C05459=1044.843,173.634,405.033,170.769,37.953,157.158
C05460=1044.836,173.349,405.060,170.766,37.951,157.157
C05461=1044.829,173.064,405.087,170.763,37.949,157.157
C05462=1044.823,172.815,405.109,170.761,37.947,157.156
C05463=1044.817,172.567,405.132,170.759,37.946,157.156
C05464=1044.810,172.318,405.156,170.756,37.945,157.156
C05465=1044.804,172.069,405.179,170.754,37.943,157.155
C05466=1044.799,171.820,405.202,170.752,37.942,157.155
C05467=1044.793,171.572,405.226,170.749,37.940,157.155
C05468=1044.787,171.323,405.249,170.747,37.938,157.154
C05469=1044.780,171.073,405.272,170.744,37.937,157.154
C05470=1044.774,170.824,405.295,170.742,37.935,157.154
C05471=1044.768,170.576,405.318,170.739,37.933,157.153
C05472=1044.762,170.327,405.341,170.737,37.932,157.153
C05473=1044.757,170.078,405.364,170.735,37.930,157.153
C05474=1044.750,169.829,405.387,170.733,37.929,157.152
C05475=1044.744,169.580,405.410,170.730,37.927,157.152
C05476=1044.738,169.331,405.433,170.728,37.926,157.151
C05477=1044.732,169.083,405.456,170.726,37.925,157.151
C05478=1044.726,168.834,405.479,170.723,37.923,157.151
C05479=1044.720,168.585,405.503,170.721,37.921,157.150
C05480=1044.714,168.336,405.526,170.719,37.920,157.150
C05481=1044.708,168.087,405.548,170.717,37.918,157.150
C05482=1044.702,167.838,405.571,170.714,37.916,157.149
C05483=1044.696,167.589,405.594,170.712,37.915,157.149
C05484=1044.690,167.341,405.617,170.709,37.913,157.149
C05485=1044.685,167.092,405.640,170.707,37.912,157.148
C05486=1044.679,166.843,405.663,170.704,37.910,157.148
C05487=1044.672,166.594,405.686,170.702,37.909,157.148
C05488=1044.666,166.345,405.709,170.700,37.907,157.147
C05489=1044.660,166.096,405.732,170.697,37.906,157.147
C05490=1044.655,165.847,405.755,170.695,37.904,157.147
C05491=1044.649,165.598,405.778,170.693,37.903,157.146
C05492=1044.642,165.350,405.800,170.691,37.901,157.146
C05493=1044.637,165.101,405.823,170.688,37.900,157.146
C05494=1044.631,164.852,405.846,170.686,37.898,157.145
C05495=1044.625,164.603,405.869,170.684,37.896,157.145
C05496=1044.619,164.354,405.892,170.682,37.895,157.145
C05497=1044.613,164.106,405.914,170.679,37.893,157.144
C05498=1044.607,163.857,405.937,170.677,37.891,157.144
C05499=1044.601,163.607,405.961,170.675,37.890,157.144
C05500=1044.595,163.358,405.984,170.672,37.889,157.143
C05501=1044.589,163.109,406.007,170.670,37.887,157.143
C05502=1044.583,162.861,406.029,170.668,37.886,157.143
C05503=1044.577,162.612,406.052,170.666,37.884,157.142
C05504=1044.572,162.363,406.075,170.663,37.883,157.142
C05505=1044.566,162.114,406.098,170.661,37.881,157.142
C05506=1044.560,161.865,406.119,170.659,37.879,157.141
C05507=1044.554,161.616,406.142,170.657,37.878,157.141
C05508=1044.548,161.367,406.165,170.654,37.876,157.140
C05509=1044.542,161.118,406.188,170.652,37.875,157.140
C05510=1044.537,160.869,406.211,170.650,37.873,157.140
C05511=1044.530,160.621,406.233,170.647,37.871,157.139
C05512=1044.525,160.372,406.256,170.645,37.870,157.139
C05513=1044.519,160.122,406.279,170.643,37.868,157.139
C05514=1044.513,159.874,406.301,170.641,37.867,157.138
C05515=1044.506,159.625,406.323,170.638,37.865,157.138
C05516=1044.501,159.376,406.346,170.636,37.864,157.138
C05517=1044.494,159.127,406.368,170.634,37.863,157.138
C05518=1044.489,158.878,406.391,170.632,37.861,157.137
C05519=1044.482,158.629,406.413,170.629,37.860,157.137
C05520=1044.476,158.380,406.435,170.627,37.858,157.137
C05521=1044.470,158.131,406.458,170.625,37.857,157.136
C05522=1044.463,157.846,406.483,170.623,37.855,157.136
C05523=1044.456,157.561,406.509,170.620,37.854,157.136
C05524=1044.449,157.275,406.534,170.617,37.852,157.135
C05525=1044.441,156.990,406.560,170.615,37.851,157.135
C05526=1044.436,156.741,406.582,170.613,37.850,157.135
C05527=1044.430,156.492,406.605,170.610,37.848,157.134
C05528=1044.423,156.243,406.626,170.608,37.847,157.134
C05529=1044.418,155.994,406.649,170.606,37.845,157.134
C05530=1044.411,155.745,406.672,170.604,37.844,157.133
C05531=1044.405,155.496,406.693,170.601,37.842,157.133
C05532=1044.400,155.248,406.716,170.599,37.841,157.133
C05533=1044.394,154.999,406.738,170.597,37.839,157.132
C05534=1044.388,154.750,406.761,170.595,37.838,157.132
C05535=1044.382,154.501,406.782,170.592,37.837,157.132
C05536=1044.375,154.252,406.804,170.590,37.835,157.131
C05537=1044.369,154.003,406.826,170.588,37.834,157.131
C05538=1044.363,153.754,406.849,170.586,37.832,157.131
C05539=1044.357,153.505,406.871,170.583,37.831,157.131
C05540=1044.351,153.256,406.893,170.581,37.829,157.130
C05541=1044.345,153.007,406.915,170.579,37.828,157.130
C05542=1044.338,152.758,406.937,170.577,37.827,157.130
C05543=1044.333,152.509,406.959,170.574,37.825,157.129
C05544=1044.326,152.260,406.982,170.572,37.824,157.129
C05545=1044.320,152.011,407.003,170.570,37.823,157.129
C05546=1044.314,151.762,407.026,170.569,37.821,157.128
C05547=1044.308,151.513,407.048,170.567,37.820,157.128
C05548=1044.302,151.264,407.069,170.564,37.819,157.128
C05549=1044.296,151.016,407.091,170.562,37.817,157.127
C05550=1044.290,150.767,407.113,170.560,37.816,157.127
C05551=1044.284,150.518,407.135,170.558,37.815,157.127
C05552=1044.278,150.269,407.158,170.555,37.813,157.126
C05553=1044.272,150.019,407.179,170.553,37.812,157.126
C05554=1044.266,149.771,407.202,170.551,37.810,157.126
C05555=1044.259,149.522,407.223,170.549,37.809,157.126
C05556=1044.253,149.272,407.245,170.546,37.808,157.125
C05557=1044.247,149.024,407.267,170.544,37.806,157.125
C05558=1044.242,148.775,407.289,170.542,37.805,157.125
C05559=1044.236,148.526,407.311,170.540,37.803,157.124
C05560=1044.230,148.277,407.332,170.538,37.802,157.124
C05561=1044.223,148.028,407.355,170.535,37.801,157.124
C05562=1044.217,147.779,407.376,170.533,37.799,157.123
C05563=1044.211,147.530,407.398,170.532,37.798,157.123
C05564=1044.205,147.280,407.420,170.530,37.797,157.123
C05565=1044.199,147.032,407.442,170.527,37.796,157.123
C05566=1044.193,146.783,407.463,170.525,37.794,157.122
C05567=1044.186,146.534,407.485,170.523,37.793,157.122
C05568=1044.180,146.285,407.507,170.521,37.792,157.122
C05569=1044.174,146.036,407.528,170.518,37.790,157.122
C05570=1044.168,145.787,407.551,170.516,37.789,157.121
C05571=1044.161,145.538,407.572,170.514,37.787,157.121
C05572=1044.156,145.289,407.593,170.512,37.786,157.121
C05573=1044.150,145.040,407.615,170.510,37.785,157.120
C05574=1044.144,144.791,407.637,170.507,37.784,157.120
C05575=1044.137,144.542,407.658,170.505,37.783,157.120
C05576=1044.131,144.293,407.680,170.503,37.781,157.119
C05577=1044.125,144.045,407.702,170.502,37.780,157.119
C05578=1044.119,143.795,407.724,170.499,37.778,157.119
C05579=1044.113,143.546,407.745,170.497,37.777,157.119
C05580=1044.107,143.297,407.767,170.495,37.775,157.118
C05581=1044.101,143.048,407.789,170.493,37.774,157.118
C05582=1044.095,142.799,407.810,170.491,37.773,157.118
C05583=1044.089,142.550,407.831,170.488,37.772,157.117
C05584=1044.082,142.301,407.852,170.486,37.771,157.117
C05585=1044.076,142.052,407.874,170.484,37.769,157.117
C05586=1044.069,141.767,407.899,170.482,37.768,157.117
C05587=1044.063,141.481,407.924,170.479,37.766,157.116
C05588=1044.056,141.195,407.949,170.477,37.765,157.116
C05589=1044.048,140.909,407.973,170.475,37.763,157.116
C05590=1044.043,140.661,407.994,170.473,37.762,157.115
C05591=1044.037,140.412,408.016,170.470,37.761,157.115
C05592=1044.030,140.162,408.037,170.468,37.759,157.115
C05593=1044.024,139.913,408.059,170.466,37.758,157.114
C05594=1044.019,139.665,408.080,170.464,37.757,157.114
C05595=1044.013,139.416,408.102,170.462,37.755,157.114
C05596=1044.006,139.166,408.123,170.459,37.754,157.114
C05597=1043.999,138.917,408.144,170.458,37.753,157.113
C05598=1043.994,138.669,408.166,170.456,37.751,157.113
C05599=1043.988,138.420,408.187,170.454,37.750,157.113
C05600=1043.982,138.170,408.209,170.451,37.749,157.112
C05601=1043.975,137.922,408.230,170.449,37.748,157.112
C05602=1043.969,137.672,408.251,170.447,37.746,157.112
C05603=1043.963,137.423,408.272,170.445,37.745,157.112
C05604=1043.957,137.174,408.294,170.443,37.744,157.111
C05605=1043.951,136.926,408.315,170.441,37.742,157.111
C05606=1043.945,136.677,408.336,170.439,37.741,157.111
C05607=1043.939,136.427,408.357,170.437,37.740,157.110
C05608=1043.933,136.179,408.378,170.435,37.739,157.110
C05609=1043.926,135.929,408.399,170.433,37.737,157.110
C05610=1043.920,135.680,408.421,170.430,37.736,157.110
C05611=1043.914,135.431,408.443,170.428,37.735,157.109
C05612=1043.908,135.182,408.463,170.426,37.734,157.109
C05613=1043.902,134.933,408.484,170.425,37.733,157.109
C05614=1043.896,134.684,408.506,170.422,37.731,157.109
C05615=1043.889,134.436,408.527,170.420,37.730,157.108
C05616=1043.884,134.186,408.547,170.418,37.729,157.108
C05617=1043.878,133.937,408.569,170.416,37.727,157.108
C05618=1043.871,133.688,408.590,170.414,37.726,157.107
C05619=1043.865,133.439,408.611,170.411,37.725,157.107
C05620=1043.860,133.190,408.632,170.410,37.724,157.107
C05621=1043.853,132.941,408.653,170.408,37.723,157.107
C05622=1043.847,132.692,408.675,170.406,37.721,157.106
C05623=1043.841,132.443,408.695,170.404,37.720,157.106
C05624=1043.834,132.194,408.716,170.401,37.718,157.106
C05625=1043.828,131.945,408.738,170.399,37.717,157.106
C05626=1043.823,131.696,408.758,170.397,37.716,157.105
C05627=1043.816,131.447,408.779,170.396,37.715,157.105
C05628=1043.811,131.198,408.800,170.394,37.714,157.105
C05629=1043.804,130.949,408.821,170.391,37.712,157.104
C05630=1043.798,130.699,408.843,170.389,37.711,157.104
C05631=1043.792,130.451,408.863,170.387,37.710,157.104
C05632=1043.785,130.202,408.884,170.385,37.709,157.104
C05633=1043.779,129.952,408.905,170.383,37.708,157.103
C05634=1043.773,129.704,408.925,170.381,37.707,157.103
C05635=1043.767,129.454,408.946,170.379,37.705,157.103
C05636=1043.760,129.205,408.967,170.377,37.704,157.103
C05637=1043.754,128.956,408.987,170.375,37.703,157.102
C05638=1043.748,128.707,409.009,170.373,37.702,157.102
C05639=1043.742,128.458,409.029,170.370,37.701,157.102
C05640=1043.735,128.209,409.050,170.368,37.699,157.102
C05641=1043.729,127.959,409.071,170.367,37.698,157.101
C05642=1043.723,127.711,409.091,170.365,37.697,157.101
C05643=1043.716,127.462,409.112,170.363,37.696,157.101
C05644=1043.711,127.213,409.132,170.360,37.695,157.101
C05645=1043.704,126.964,409.153,170.358,37.693,157.100
C05646=1043.698,126.714,409.174,170.356,37.692,157.100
C05647=1043.692,126.466,409.195,170.354,37.691,157.100
C05648=1043.685,126.216,409.215,170.353,37.690,157.100
C05649=1043.680,125.967,409.236,170.350,37.689,157.099
C05650=1043.672,125.681,409.260,170.348,37.687,157.099
C05651=1043.665,125.396,409.284,170.346,37.686,157.099
C05652=1043.658,125.110,409.308,170.343,37.685,157.098
C05653=1043.651,124.824,409.331,170.341,37.683,157.098
C05654=1043.645,124.575,409.351,170.339,37.682,157.098
C05655=1043.639,124.325,409.372,170.337,37.681,157.098
C05656=1043.633,124.077,409.393,170.335,37.680,157.097
C05657=1043.626,123.828,409.413,170.333,37.679,157.097
C05658=1043.620,123.578,409.434,170.331,37.677,157.097
C05659=1043.614,123.330,409.455,170.328,37.676,157.097
C05660=1043.607,123.080,409.475,170.327,37.675,157.096
C05661=1043.602,122.831,409.496,170.325,37.674,157.096
C05662=1043.595,122.582,409.516,170.323,37.673,157.096
C05663=1043.589,122.333,409.537,170.321,37.671,157.096
C05664=1043.583,122.085,409.557,170.318,37.670,157.095
C05665=1043.577,121.835,409.577,170.317,37.669,157.095
C05666=1043.571,121.587,409.598,170.315,37.668,157.095
C05667=1043.564,121.337,409.618,170.313,37.667,157.095
C05668=1043.559,121.088,409.639,170.311,37.665,157.094
C05669=1043.553,120.838,409.659,170.308,37.664,157.094
C05670=1043.547,120.590,409.679,170.307,37.663,157.094
C05671=1043.540,120.340,409.701,170.305,37.662,157.093
C05672=1043.534,120.092,409.721,170.303,37.661,157.093
C05673=1043.528,119.842,409.741,170.301,37.659,157.093
C05674=1043.523,119.593,409.762,170.298,37.658,157.093
C05675=1043.516,119.345,409.782,170.297,37.657,157.092
C05676=1043.510,119.095,409.803,170.295,37.656,157.092
C05677=1043.504,118.846,409.823,170.293,37.655,157.092
C05678=1043.498,118.597,409.844,170.291,37.653,157.092
C05679=1043.492,118.348,409.864,170.288,37.652,157.091
C05680=1043.485,118.098,409.884,170.287,37.651,157.091
C05681=1043.480,117.849,409.904,170.285,37.650,157.091
C05682=1043.474,117.601,409.925,170.283,37.649,157.091
C05683=1043.467,117.351,409.945,170.281,37.647,157.090
C05684=1043.461,117.103,409.965,170.280,37.646,157.090
C05685=1043.456,116.854,409.986,170.277,37.645,157.090
C05686=1043.449,116.604,410.006,170.275,37.644,157.090
C05687=1043.443,116.355,410.026,170.273,37.643,157.089
C05688=1043.437,116.105,410.047,170.271,37.641,157.089
C05689=1043.431,115.857,410.067,170.269,37.640,157.089
C05690=1043.425,115.608,410.087,170.267,37.638,157.088
C05691=1043.419,115.358,410.107,170.265,37.637,157.088
C05692=1043.413,115.110,410.129,170.263,37.636,157.088
C05693=1043.407,114.861,410.149,170.262,37.635,157.088
C05694=1043.401,114.611,410.169,170.259,37.634,157.087
C05695=1043.395,114.363,410.189,170.257,37.632,157.087
C05696=1043.389,114.113,410.209,170.255,37.631,157.087
C05697=1043.383,113.864,410.230,170.254,37.630,157.087
C05698=1043.377,113.615,410.250,170.252,37.629,157.086
C05699=1043.371,113.366,410.270,170.250,37.628,157.086
C05700=1043.364,113.117,410.290,170.247,37.626,157.086
C05701=1043.358,112.868,410.310,170.246,37.625,157.086
C05702=1043.353,112.619,410.329,170.244,37.624,157.085
C05703=1043.346,112.369,410.350,170.242,37.623,157.085
C05704=1043.340,112.120,410.370,170.240,37.622,157.085
C05705=1043.333,111.871,410.390,170.237,37.621,157.085
C05706=1043.327,111.622,410.410,170.236,37.620,157.085
C05707=1043.321,111.373,410.430,170.234,37.619,157.084
C05708=1043.315,111.124,410.450,170.232,37.617,157.084
C05709=1043.309,110.875,410.470,170.230,37.616,157.084
C05710=1043.303,110.626,410.490,170.228,37.615,157.083
C05711=1043.296,110.376,410.510,170.226,37.614,157.083
C05712=1043.290,110.127,410.530,170.224,37.613,157.083
C05713=1043.284,109.878,410.550,170.222,37.611,157.083
C05714=1043.278,109.592,410.572,170.220,37.610,157.082
C05715=1043.270,109.306,410.595,170.218,37.609,157.082
C05716=1043.263,109.020,410.618,170.215,37.608,157.082
C05717=1043.256,108.734,410.640,170.213,37.607,157.082
C05718=1043.250,108.485,410.660,170.211,37.605,157.081
C05719=1043.243,108.236,410.681,170.209,37.604,157.081
C05720=1043.237,107.986,410.700,170.208,37.603,157.081
C05721=1043.231,107.737,410.720,170.205,37.602,157.081
C05722=1043.224,107.488,410.740,170.203,37.601,157.081
C05723=1043.218,107.239,410.760,170.201,37.600,157.080
C05724=1043.212,106.990,410.779,170.200,37.599,157.080
C05725=1043.206,106.741,410.799,170.198,37.598,157.080
C05726=1043.200,106.492,410.819,170.195,37.596,157.079
C05727=1043.194,106.243,410.839,170.193,37.595,157.079
C05728=1043.188,105.993,410.858,170.192,37.594,157.079
C05729=1043.181,105.745,410.878,170.190,37.593,157.079
C05730=1043.175,105.495,410.898,170.188,37.592,157.079
C05731=1043.169,105.246,410.917,170.186,37.591,157.078
C05732=1043.163,104.997,410.937,170.183,37.590,157.078
C05733=1043.157,104.748,410.957,170.182,37.589,157.078
C05734=1043.151,104.498,410.977,170.180,37.587,157.078
C05735=1043.144,104.250,410.996,170.178,37.586,157.077
C05736=1043.138,104.000,411.015,170.176,37.585,157.077
C05737=1043.132,103.751,411.035,170.174,37.584,157.077
C05738=1043.126,103.502,411.056,170.172,37.583,157.077
C05739=1043.120,103.253,411.075,170.170,37.582,157.076
C05740=1043.113,103.004,411.094,170.168,37.581,157.076
C05741=1043.108,102.755,411.114,170.167,37.580,157.076
C05742=1043.102,102.506,411.134,170.165,37.578,157.076
C05743=1043.095,102.256,411.154,170.162,37.577,157.075
C05744=1043.089,102.007,411.173,170.160,37.576,157.075
C05745=1043.083,101.758,411.192,170.159,37.575,157.075
C05746=1043.077,101.509,411.212,170.157,37.574,157.075
C05747=1043.071,101.260,411.232,170.155,37.572,157.074
C05748=1043.065,101.010,411.251,170.154,37.572,157.074
C05749=1043.059,100.761,411.271,170.151,37.571,157.074
C05750=1043.052,100.512,411.290,170.149,37.569,157.074
C05751=1043.046,100.263,411.310,170.147,37.568,157.073
C05752=1043.041,100.014,411.329,170.146,37.567,157.073
C05753=1043.033,99.765,411.349,170.144,37.566,157.073
C05754=1043.028,99.515,411.368,170.142,37.565,157.073
C05755=1043.021,99.267,411.387,170.139,37.564,157.073
C05756=1043.015,99.017,411.407,170.137,37.563,157.072
C05757=1043.008,98.769,411.426,170.136,37.562,157.072
C05758=1043.002,98.519,411.446,170.134,37.561,157.072
C05759=1042.996,98.269,411.465,170.132,37.560,157.072
C05760=1042.990,98.021,411.484,170.129,37.559,157.071
C05761=1042.984,97.771,411.504,170.128,37.557,157.071
C05762=1042.977,97.523,411.523,170.126,37.556,157.071
C05763=1042.972,97.273,411.542,170.124,37.556,157.071
C05764=1042.965,97.023,411.561,170.122,37.554,157.071
C05765=1042.959,96.775,411.581,170.121,37.553,157.070
C05766=1042.952,96.525,411.600,170.118,37.552,157.070
C05767=1042.946,96.276,411.619,170.116,37.551,157.070
C05768=1042.940,96.028,411.638,170.114,37.550,157.070
C05769=1042.934,95.778,411.658,170.113,37.549,157.069
C05770=1042.928,95.529,411.677,170.111,37.548,157.069
C05771=1042.921,95.279,411.697,170.109,37.547,157.069
C05772=1042.915,95.030,411.716,170.106,37.545,157.069
C05773=1042.909,94.781,411.734,170.105,37.545,157.069
C05774=1042.903,94.532,411.754,170.103,37.544,157.068
C05775=1042.896,94.283,411.773,170.101,37.542,157.068
C05776=1042.891,94.034,411.792,170.099,37.541,157.068
C05777=1042.884,93.784,411.811,170.098,37.540,157.067
C05778=1042.877,93.499,411.833,170.095,37.539,157.067
C05779=1042.871,93.212,411.856,170.093,37.537,157.067
C05780=1042.863,92.926,411.878,170.091,37.536,157.067
C05781=1042.856,92.640,411.899,170.089,37.535,157.066
C05782=1042.850,92.391,411.918,170.087,37.534,157.066
C05783=1042.844,92.142,411.938,170.084,37.533,157.066
C05784=1042.837,91.893,411.957,170.083,37.532,157.066
C05785=1042.831,91.644,411.976,170.081,37.531,157.066
C05786=1042.825,91.394,411.995,170.079,37.530,157.065
C05787=1042.819,91.145,412.014,170.077,37.528,157.065
C05788=1042.813,90.897,412.033,170.076,37.527,157.065
C05789=1042.807,90.647,412.052,170.073,37.526,157.065
C05790=1042.800,90.398,412.071,170.071,37.525,157.064
C05791=1042.795,90.149,412.090,170.070,37.524,157.064
C05792=1042.788,89.899,412.109,170.068,37.523,157.064
C05793=1042.782,89.650,412.128,170.066,37.522,157.064
C05794=1042.776,89.400,412.147,170.064,37.521,157.064
C05795=1042.769,89.151,412.166,170.061,37.520,157.063
C05796=1042.763,88.902,412.185,170.060,37.519,157.063
C05797=1042.756,88.653,412.203,170.058,37.518,157.063
C05798=1042.750,88.404,412.223,170.056,37.517,157.063
C05799=1042.744,88.155,412.242,170.054,37.516,157.062
C05800=1042.737,87.906,412.260,170.053,37.515,157.062
C05801=1042.731,87.657,412.279,170.050,37.514,157.062
C05802=1042.725,87.407,412.298,170.048,37.513,157.062
C05803=1042.719,87.158,412.317,170.046,37.512,157.061
C05804=1042.713,86.909,412.336,170.045,37.511,157.061
C05805=1042.706,86.660,412.354,170.043,37.510,157.061
C05806=1042.700,86.410,412.374,170.041,37.509,157.061
C05807=1042.694,86.161,412.392,170.039,37.507,157.061
C05808=1042.688,85.912,412.411,170.037,37.507,157.060
C05809=1042.681,85.663,412.430,170.035,37.506,157.060
C05810=1042.675,85.414,412.448,170.033,37.504,157.060
C05811=1042.669,85.164,412.467,170.032,37.504,157.060
C05812=1042.663,84.915,412.485,170.030,37.503,157.060
C05813=1042.656,84.666,412.504,170.028,37.501,157.059
C05814=1042.650,84.416,412.523,170.025,37.500,157.059
C05815=1042.644,84.167,412.542,170.024,37.499,157.059
C05816=1042.638,83.918,412.561,170.022,37.498,157.059
C05817=1042.632,83.669,412.579,170.020,37.497,157.058
C05818=1042.625,83.420,412.598,170.018,37.496,157.058
C05819=1042.619,83.171,412.616,170.017,37.495,157.058
C05820=1042.613,82.921,412.636,170.014,37.494,157.058
C05821=1042.607,82.672,412.654,170.012,37.493,157.058
C05822=1042.600,82.423,412.673,170.010,37.492,157.057
C05823=1042.594,82.173,412.691,170.009,37.491,157.057
C05824=1042.588,81.924,412.710,170.007,37.490,157.057
C05825=1042.582,81.675,412.729,170.005,37.489,157.057
C05826=1042.575,81.425,412.747,170.003,37.487,157.056
C05827=1042.570,81.177,412.766,170.001,37.487,157.056
C05828=1042.563,80.928,412.784,169.999,37.486,157.056
C05829=1042.557,80.678,412.802,169.997,37.484,157.056
C05830=1042.551,80.429,412.822,169.996,37.483,157.056
C05831=1042.545,80.180,412.840,169.994,37.483,157.055
C05832=1042.539,79.931,412.859,169.991,37.481,157.055
C05833=1042.532,79.681,412.878,169.990,37.480,157.055
C05834=1042.526,79.432,412.895,169.988,37.479,157.055
C05835=1042.520,79.182,412.915,169.986,37.478,157.055
C05836=1042.514,78.933,412.933,169.984,37.477,157.054
C05837=1042.508,78.685,412.952,169.983,37.476,157.054
C05838=1042.502,78.436,412.970,169.980,37.475,157.054
C05839=1042.496,78.186,412.988,169.978,37.474,157.054
C05840=1042.489,77.937,413.007,169.976,37.473,157.053
C05841=1042.483,77.688,413.026,169.975,37.472,157.053
C05842=1042.476,77.401,413.046,169.973,37.470,157.053
C05843=1042.469,77.115,413.067,169.971,37.469,157.053
C05844=1042.461,76.829,413.089,169.968,37.468,157.052
C05845=1042.454,76.543,413.110,169.966,37.467,157.052
C05846=1042.448,76.295,413.128,169.964,37.466,157.052
C05847=1042.442,76.045,413.146,169.962,37.465,157.052
C05848=1042.435,75.796,413.165,169.961,37.464,157.051
C05849=1042.429,75.546,413.183,169.959,37.463,157.051
C05850=1042.423,75.297,413.201,169.956,37.462,157.051
C05851=1042.416,75.048,413.220,169.954,37.461,157.051
C05852=1042.410,74.798,413.238,169.953,37.460,157.051
C05853=1042.404,74.549,413.256,169.951,37.459,157.050
C05854=1042.398,74.300,413.274,169.949,37.458,157.050
C05855=1042.392,74.051,413.293,169.947,37.457,157.050
C05856=1042.385,73.802,413.311,169.946,37.456,157.050
C05857=1042.379,73.552,413.329,169.943,37.455,157.050
C05858=1042.372,73.303,413.347,169.941,37.454,157.049
C05859=1042.366,73.053,413.365,169.939,37.453,157.049
C05860=1042.360,72.805,413.384,169.938,37.452,157.049
C05861=1042.354,72.555,413.401,169.936,37.451,157.049
C05862=1042.348,72.306,413.420,169.934,37.450,157.049
C05863=1042.341,72.056,413.438,169.931,37.449,157.048
C05864=1042.335,71.807,413.457,169.930,37.448,157.048
C05865=1042.329,71.558,413.474,169.928,37.447,157.048
C05866=1042.323,71.309,413.493,169.926,37.446,157.048
C05867=1042.317,71.059,413.511,169.925,37.445,157.048
C05868=1042.310,70.810,413.529,169.923,37.444,157.047
C05869=1042.304,70.561,413.547,169.920,37.443,157.047
C05870=1042.298,70.312,413.565,169.918,37.442,157.047
C05871=1042.292,70.062,413.583,169.917,37.441,157.047
C05872=1042.285,69.813,413.602,169.915,37.440,157.046
C05873=1042.279,69.564,413.620,169.913,37.439,157.046
C05874=1042.273,69.314,413.638,169.911,37.438,157.046
C05875=1042.266,69.066,413.655,169.910,37.437,157.046
C05876=1042.260,68.816,413.673,169.907,37.436,157.046
C05877=1042.254,68.567,413.692,169.905,37.435,157.045
C05878=1042.248,68.317,413.710,169.903,37.434,157.045
C05879=1042.242,68.068,413.727,169.902,37.433,157.045
C05880=1042.235,67.819,413.745,169.900,37.432,157.045
C05881=1042.229,67.570,413.763,169.898,37.431,157.045
C05882=1042.223,67.320,413.781,169.896,37.430,157.044
C05883=1042.216,67.071,413.799,169.894,37.429,157.044
C05884=1042.210,66.822,413.817,169.892,37.428,157.044
C05885=1042.204,66.572,413.835,169.890,37.427,157.044
C05886=1042.198,66.323,413.853,169.888,37.426,157.044
C05887=1042.191,66.074,413.871,169.887,37.425,157.043
C05888=1042.185,65.825,413.888,169.885,37.424,157.043
C05889=1042.179,65.576,413.907,169.883,37.423,157.043
C05890=1042.172,65.326,413.924,169.880,37.422,157.043
C05891=1042.166,65.077,413.942,169.879,37.421,157.043
C05892=1042.160,64.827,413.960,169.877,37.420,157.042
C05893=1042.153,64.579,413.978,169.875,37.419,157.042
C05894=1042.147,64.329,413.996,169.873,37.418,157.042
C05895=1042.142,64.080,414.013,169.872,37.417,157.042
C05896=1042.135,63.830,414.031,169.869,37.416,157.041
C05897=1042.129,63.581,414.049,169.867,37.415,157.041
C05898=1042.121,63.332,414.067,169.865,37.415,157.041
C05899=1042.116,63.083,414.084,169.864,37.413,157.041
C05900=1042.109,62.833,414.102,169.862,37.413,157.041
C05901=1042.102,62.584,414.119,169.860,37.412,157.041
C05902=1042.096,62.334,414.137,169.858,37.411,157.040
C05903=1042.090,62.085,414.154,169.857,37.410,157.040
C05904=1042.083,61.836,414.173,169.854,37.409,157.040
C05905=1042.076,61.587,414.190,169.852,37.408,157.040
C05906=1042.070,61.301,414.210,169.850,37.407,157.040
C05907=1042.062,61.014,414.230,169.848,37.406,157.039
C05908=1042.055,60.728,414.250,169.846,37.405,157.039
C05909=1042.047,60.442,414.270,169.844,37.404,157.039
C05910=1042.041,60.192,414.288,169.842,37.403,157.039
C05911=1042.035,59.943,414.305,169.839,37.402,157.039
C05912=1042.028,59.694,414.323,169.838,37.401,157.038
C05913=1042.022,59.444,414.341,169.836,37.400,157.038
C05914=1042.016,59.195,414.358,169.834,37.400,157.038
C05915=1042.009,58.946,414.375,169.832,37.398,157.038
C05916=1042.003,58.696,414.393,169.830,37.398,157.038
C05917=1041.996,58.447,414.410,169.829,37.397,157.037
C05918=1041.990,58.198,414.427,169.826,37.396,157.037
C05919=1041.984,57.948,414.445,169.824,37.395,157.037
C05920=1041.977,57.700,414.462,169.822,37.394,157.037
C05921=1041.971,57.450,414.480,169.821,37.393,157.037
C05922=1041.964,57.200,414.497,169.819,37.392,157.037
C05923=1041.958,56.952,414.514,169.817,37.391,157.036
C05924=1041.952,56.702,414.532,169.815,37.391,157.036
C05925=1041.945,56.452,414.550,169.813,37.389,157.036
C05926=1041.940,56.203,414.567,169.811,37.389,157.036
C05927=1041.933,55.954,414.584,169.809,37.387,157.036
C05928=1041.926,55.705,414.602,169.807,37.387,157.035
C05929=1041.920,55.455,414.619,169.805,37.386,157.035
C05930=1041.914,55.206,414.637,169.804,37.385,157.035
C05931=1041.907,54.957,414.654,169.802,37.384,157.035
C05932=1041.901,54.708,414.672,169.799,37.383,157.035
C05933=1041.894,54.458,414.689,169.797,37.382,157.034
C05934=1041.889,54.209,414.706,169.796,37.381,157.034
C05935=1041.882,53.959,414.723,169.794,37.380,157.034
C05936=1041.876,53.710,414.740,169.792,37.379,157.034
C05937=1041.870,53.461,414.758,169.790,37.378,157.034
C05938=1041.864,53.212,414.775,169.789,37.377,157.033
C05939=1041.857,52.962,414.792,169.787,37.377,157.033
C05940=1041.851,52.713,414.810,169.784,37.375,157.033
C05941=1041.844,52.464,414.827,169.782,37.375,157.033
C05942=1041.839,52.214,414.844,169.780,37.373,157.033
C05943=1041.832,51.965,414.861,169.779,37.372,157.032
C05944=1041.825,51.715,414.879,169.777,37.372,157.032
C05945=1041.820,51.466,414.896,169.775,37.370,157.032
C05946=1041.813,51.217,414.914,169.773,37.370,157.032
C05947=1041.807,50.968,414.931,169.771,37.369,157.032
C05948=1041.801,50.718,414.948,169.769,37.368,157.032
C05949=1041.795,50.469,414.965,169.767,37.367,157.031
C05950=1041.788,50.220,414.982,169.765,37.366,157.031
C05951=1041.782,49.971,415.000,169.764,37.365,157.031
C05952=1041.776,49.721,415.016,169.762,37.364,157.031
C05953=1041.770,49.472,415.033,169.760,37.363,157.031
C05954=1041.763,49.222,415.051,169.757,37.362,157.030
C05955=1041.757,48.973,415.068,169.756,37.361,157.030
C05956=1041.751,48.723,415.085,169.754,37.360,157.030
C05957=1041.745,48.474,415.102,169.752,37.359,157.030
C05958=1041.738,48.225,415.120,169.750,37.358,157.029
C05959=1041.732,47.976,415.137,169.749,37.357,157.029
C05960=1041.726,47.726,415.154,169.747,37.356,157.029
C05961=1041.720,47.477,415.171,169.744,37.355,157.029
C05962=1041.713,47.228,415.188,169.742,37.355,157.029
C05963=1041.708,46.978,415.205,169.740,37.353,157.028
C05964=1041.702,46.729,415.222,169.739,37.352,157.028
C05965=1041.695,46.480,415.239,169.737,37.352,157.028
C05966=1041.690,46.230,415.256,169.735,37.350,157.028
C05967=1041.683,45.981,415.274,169.733,37.350,157.028
C05968=1041.676,45.732,415.291,169.731,37.348,157.027
C05969=1041.671,45.482,415.308,169.729,37.347,157.027
C05970=1041.663,45.196,415.327,169.727,37.347,157.027
C05971=1041.656,44.909,415.346,169.725,37.345,157.027
C05972=1041.649,44.623,415.367,169.723,37.344,157.027
C05973=1041.642,44.336,415.386,169.721,37.343,157.026
C05974=1041.635,44.087,415.403,169.718,37.342,157.026
C05975=1041.630,43.837,415.420,169.716,37.341,157.026
C05976=1041.624,43.588,415.437,169.715,37.340,157.026
C05977=1041.617,43.338,415.454,169.713,37.339,157.026
C05978=1041.611,43.090,415.471,169.711,37.338,157.025
C05979=1041.604,42.840,415.487,169.709,37.337,157.025
C05980=1041.599,42.591,415.505,169.707,37.336,157.025
C05981=1041.593,42.341,415.521,169.705,37.336,157.025
C05982=1041.586,42.092,415.538,169.703,37.334,157.025
C05983=1041.580,41.842,415.555,169.701,37.334,157.024
C05984=1041.573,41.593,415.572,169.699,37.333,157.024
C05985=1041.567,41.344,415.588,169.697,37.332,157.024
C05986=1041.561,41.095,415.605,169.696,37.331,157.024
C05987=1041.554,40.845,415.622,169.694,37.330,157.024
C05988=1041.548,40.596,415.639,169.692,37.329,157.023
C05989=1041.542,40.346,415.656,169.689,37.328,157.023
C05990=1041.536,40.097,415.672,169.687,37.328,157.023
C05991=1041.529,39.848,415.689,169.686,37.327,157.023
C05992=1041.523,39.598,415.705,169.684,37.326,157.023
C05993=1041.517,39.349,415.722,169.682,37.325,157.023
C05994=1041.511,39.100,415.739,169.680,37.324,157.022
C05995=1041.504,38.851,415.756,169.678,37.323,157.022
C05996=1041.498,38.601,415.772,169.677,37.322,157.022
C05997=1041.491,38.351,415.789,169.674,37.321,157.022
C05998=1041.485,38.102,415.806,169.672,37.320,157.022
C05999=1041.479,37.853,415.822,169.670,37.319,157.021
C06000=1041.473,37.603,415.839,169.668,37.319,157.021
C06001=1041.466,37.354,415.856,169.667,37.317,157.021
C06002=1041.460,37.105,415.872,169.665,37.317,157.021
C06003=1041.454,36.855,415.889,169.663,37.316,157.021
C06004=1041.447,36.606,415.906,169.660,37.315,157.021
C06005=1041.442,36.357,415.922,169.658,37.314,157.020
C06006=1041.435,36.107,415.938,169.657,37.313,157.020
C06007=1041.428,35.858,415.954,169.655,37.312,157.020
C06008=1041.422,35.609,415.971,169.653,37.312,157.020
C06009=1041.415,35.359,415.988,169.651,37.311,157.020
C06010=1041.410,35.110,416.004,169.649,37.310,157.020
C06011=1041.404,34.860,416.020,169.647,37.309,157.019
C06012=1041.397,34.611,416.037,169.645,37.308,157.019
C06013=1041.390,34.362,416.053,169.643,37.308,157.019
C06014=1041.384,34.112,416.069,169.641,37.306,157.019
C06015=1041.378,33.862,416.086,169.639,37.306,157.019
C06016=1041.372,33.613,416.102,169.637,37.305,157.018
C06017=1041.365,33.364,416.119,169.635,37.304,157.018
C06018=1041.358,33.115,416.135,169.634,37.303,157.018
C06019=1041.352,32.865,416.152,169.632,37.302,157.018
C06020=1041.346,32.616,416.168,169.629,37.302,157.018
C06021=1041.340,32.366,416.184,169.627,37.300,157.018
C06022=1041.333,32.117,416.201,169.625,37.300,157.017
C06023=1041.327,31.868,416.217,169.624,37.299,157.017
C06024=1041.321,31.619,416.233,169.622,37.298,157.017
C06025=1041.314,31.369,416.250,169.620,37.297,157.017
C06026=1041.308,31.119,416.266,169.618,37.296,157.017
C06027=1041.302,30.870,416.282,169.616,37.295,157.017
C06028=1041.296,30.621,416.298,169.614,37.295,157.016
C06029=1041.289,30.371,416.315,169.612,37.294,157.016
C06030=1041.283,30.122,416.332,169.610,37.293,157.016
C06031=1041.277,29.873,416.348,169.608,37.292,157.016
C06032=1041.270,29.624,416.364,169.606,37.291,157.016
C06033=1041.264,29.374,416.380,169.604,37.291,157.016
C06034=1041.257,29.086,416.399,169.602,37.289,157.015
C06035=1041.250,28.800,416.417,169.600,37.288,157.015
C06036=1041.242,28.514,416.436,169.597,37.288,157.015
C06037=1041.235,28.228,416.455,169.595,37.286,157.015
C06038=1041.229,27.978,416.471,169.593,37.286,157.015
C06039=1041.223,27.728,416.488,169.591,37.285,157.014
C06040=1041.216,27.479,416.503,169.589,37.284,157.014
C06041=1041.210,27.229,416.519,169.587,37.283,157.014
C06042=1041.203,26.980,416.534,169.586,37.283,157.014
C06043=1041.197,26.730,416.551,169.584,37.281,157.014
C06044=1041.191,26.481,416.567,169.581,37.281,157.014
C06045=1041.184,26.232,416.583,169.579,37.280,157.013
C06046=1041.178,25.983,416.599,169.577,37.279,157.013
C06047=1041.172,25.733,416.615,169.575,37.278,157.013
C06048=1041.165,25.483,416.632,169.573,37.278,157.013
C06049=1041.159,25.234,416.648,169.572,37.277,157.013
C06050=1041.152,24.985,416.663,169.570,37.276,157.013
C06051=1041.147,24.736,416.680,169.568,37.275,157.012
C06052=1041.140,24.487,416.695,169.565,37.274,157.012
C06053=1041.133,24.237,416.712,169.563,37.273,157.012
C06054=1041.127,23.987,416.727,169.561,37.273,157.012
C06055=1041.121,23.738,416.743,169.559,37.272,157.012
C06056=1041.114,23.489,416.759,169.557,37.271,157.012
C06057=1041.108,23.239,416.775,169.556,37.270,157.011
C06058=1041.102,22.990,416.791,169.554,37.269,157.011
C06059=1041.095,22.740,416.807,169.552,37.269,157.011
C06060=1041.089,22.490,416.823,169.550,37.268,157.011
C06061=1041.083,22.241,416.839,169.548,37.267,157.011
C06062=1041.077,21.992,416.855,169.545,37.266,157.011
C06063=1041.070,21.743,416.871,169.543,37.266,157.010
C06064=1041.064,21.493,416.887,169.542,37.265,157.010
C06065=1041.058,21.244,416.902,169.540,37.264,157.010
C06066=1041.052,20.994,416.918,169.538,37.263,157.010
C06067=1041.045,20.745,416.934,169.536,37.263,157.010
C06068=1041.039,20.495,416.950,169.534,37.261,157.010
C06069=1041.032,20.246,416.966,169.532,37.261,157.009
C06070=1041.026,19.996,416.981,169.529,37.260,157.009
C06071=1041.020,19.747,416.997,169.527,37.259,157.009
C06072=1041.014,19.498,417.013,169.526,37.258,157.009
C06073=1041.007,19.248,417.028,169.524,37.258,157.009
C06074=1041.001,18.999,417.045,169.522,37.257,157.009
C06075=1040.995,18.750,417.060,169.520,37.256,157.008
C06076=1040.988,18.500,417.075,169.518,37.255,157.008
C06077=1040.982,18.250,417.092,169.516,37.255,157.008
C06078=1040.975,18.001,417.107,169.513,37.253,157.008
C06079=1040.969,17.751,417.123,169.511,37.253,157.008
C06080=1040.963,17.502,417.139,169.509,37.252,157.008
C06081=1040.956,17.253,417.154,169.508,37.252,157.008
C06082=1040.950,17.003,417.170,169.506,37.250,157.007
C06083=1040.944,16.754,417.186,169.504,37.250,157.007
C06084=1040.938,16.505,417.202,169.502,37.249,157.007
C06085=1040.931,16.255,417.217,169.500,37.249,157.007
C06086=1040.925,16.006,417.232,169.498,37.247,157.007
C06087=1040.919,15.756,417.248,169.496,37.247,157.007
C06088=1040.912,15.507,417.264,169.493,37.246,157.006
C06089=1040.906,15.258,417.279,169.491,37.245,157.006
C06090=1040.900,15.008,417.295,169.489,37.244,157.006
C06091=1040.893,14.759,417.310,169.488,37.244,157.006
C06092=1040.888,14.509,417.326,169.486,37.243,157.006
C06093=1040.881,14.260,417.342,169.484,37.242,157.006
C06094=1040.874,14.010,417.357,169.482,37.241,157.005
C06095=1040.868,13.761,417.372,169.480,37.241,157.005
C06096=1040.862,13.511,417.388,169.478,37.240,157.005
C06097=1040.855,13.262,417.404,169.475,37.239,157.005
C06098=1040.845,12.862,417.428,169.472,37.238,157.005
C06099=1040.834,12.462,417.452,169.469,37.237,157.005
C06100=1040.824,12.062,417.477,169.466,37.236,157.004
C06101=1040.814,11.662,417.502,169.463,37.235,157.004
C06102=1040.807,11.412,417.517,169.461,37.234,157.004
C06103=1040.801,11.163,417.532,169.459,37.233,157.004
C06104=1040.794,10.914,417.547,169.457,37.233,157.004
C06105=1040.788,10.665,417.563,169.454,37.232,157.004
C06106=1040.782,10.415,417.579,169.452,37.231,157.003
C06107=1040.776,10.165,417.594,169.450,37.231,157.003
C06108=1040.769,9.916,417.609,169.448,37.230,157.003
C06109=1040.763,9.666,417.624,169.446,37.229,157.003
C06110=1040.756,9.417,417.640,169.444,37.228,157.003
C06111=1040.750,9.168,417.655,169.442,37.228,157.003
C06112=1040.743,8.918,417.670,169.440,37.227,157.003
C06113=1040.736,8.669,417.685,169.438,37.227,157.002
C06114=1040.730,8.419,417.700,169.436,37.226,157.002
C06115=1040.724,8.169,417.716,169.433,37.225,157.002
C06116=1040.718,7.920,417.731,169.431,37.225,157.002
C06117=1040.711,7.671,417.746,169.429,37.224,157.002
C06118=1040.705,7.421,417.761,169.428,37.223,157.002
C06119=1040.699,7.171,417.776,169.426,37.222,157.002
C06120=1040.692,6.922,417.792,169.424,37.222,157.001
C06121=1040.685,6.673,417.807,169.422,37.221,157.001
C06122=1040.680,6.424,417.822,169.420,37.221,157.001
C06123=1040.673,6.174,417.836,169.418,37.219,157.001
C06124=1040.667,5.925,417.852,169.415,37.219,157.001
C06125=1040.660,5.675,417.867,169.413,37.218,157.001
C06126=1040.655,5.425,417.883,169.411,37.217,157.001
C06127=1040.648,5.176,417.898,169.409,37.217,157.000
C06128=1040.642,4.927,417.913,169.407,37.216,157.000
C06129=1040.635,4.677,417.928,169.405,37.216,157.000
C06130=1040.629,4.427,417.943,169.403,37.214,157.000
C06131=1040.623,4.178,417.958,169.401,37.214,157.000
C06132=1040.617,3.929,417.973,169.399,37.213,157.000
C06133=1040.610,3.680,417.988,169.397,37.213,157.000
C06134=1040.604,3.430,418.003,169.395,37.212,156.999
C06135=1040.597,3.180,418.018,169.392,37.211,156.999
C06136=1040.591,2.931,418.033,169.390,37.210,156.999
C06137=1040.584,2.681,418.048,169.388,37.210,156.999
C06138=1040.579,2.432,418.063,169.386,37.209,156.999
C06139=1040.572,2.183,418.078,169.384,37.208,156.999
C06140=1040.566,1.933,418.093,169.382,37.208,156.999
C06141=1040.560,1.683,418.109,169.380,37.207,156.998
C06142=1040.554,1.434,418.124,169.378,37.207,156.998
C06143=1040.548,1.185,418.138,169.377,37.205,156.998
C06144=1040.541,0.935,418.153,169.374,37.205,156.998
C06145=1040.535,0.685,418.168,169.372,37.204,156.998
C06146=1040.529,0.436,418.183,169.370,37.203,156.998
C06147=1040.522,0.186,418.198,169.368,37.203,156.998
C06148=1040.516,-0.063,418.213,169.366,37.202,156.997
C06149=1040.510,-0.312,418.228,169.364,37.201,156.997
C06150=1040.503,-0.562,418.243,169.362,37.200,156.997
C06151=1040.497,-0.811,418.258,169.360,37.200,156.997
C06152=1040.491,-1.061,418.273,169.358,37.199,156.997
C06153=1040.485,-1.310,418.288,169.356,37.199,156.997
C06154=1040.475,-1.694,418.311,169.352,37.197,156.996
C06155=1040.466,-2.079,418.334,169.349,37.196,156.996
C06156=1040.456,-2.463,418.356,169.346,37.195,156.996
C06157=1040.447,-2.848,418.379,169.343,37.194,156.996
C06158=1040.439,-3.131,418.396,169.340,37.193,156.996
C06159=1040.432,-3.414,418.413,169.338,37.192,156.995
C06160=1040.425,-3.698,418.429,169.336,37.192,156.995
C06161=1040.417,-3.981,418.446,169.333,37.191,156.995
C06162=1040.412,-4.231,418.460,169.331,37.191,156.995
C06163=1040.405,-4.480,418.475,169.328,37.190,156.995
C06164=1040.399,-4.730,418.490,169.326,37.189,156.995
C06165=1040.392,-4.979,418.505,169.324,37.189,156.995
C06166=1040.386,-5.228,418.519,169.322,37.188,156.995
C06167=1040.380,-5.478,418.534,169.320,37.188,156.994
C06168=1040.373,-5.727,418.548,169.318,37.187,156.994
C06169=1040.367,-5.978,418.563,169.316,37.186,156.994
C06170=1040.361,-6.227,418.577,169.314,37.186,156.994
C06171=1040.354,-6.476,418.592,169.312,37.185,156.994
C06172=1040.347,-6.726,418.607,169.310,37.185,156.994
C06173=1040.341,-6.975,418.621,169.308,37.184,156.994
C06174=1040.335,-7.225,418.635,169.305,37.183,156.994
C06175=1040.328,-7.474,418.650,169.303,37.183,156.993
C06176=1040.322,-7.724,418.665,169.301,37.182,156.993
C06177=1040.316,-7.973,418.679,169.299,37.182,156.993
C06178=1040.309,-8.223,418.693,169.297,37.181,156.993
C06179=1040.303,-8.472,418.708,169.295,37.180,156.993
C06180=1040.297,-8.722,418.723,169.293,37.180,156.993
C06181=1040.291,-8.971,418.737,169.291,37.179,156.993
C06182=1040.284,-9.221,418.751,169.289,37.179,156.993
C06183=1040.278,-9.471,418.766,169.287,37.178,156.992
C06184=1040.272,-9.720,418.781,169.285,37.177,156.992
C06185=1040.265,-9.970,418.794,169.282,37.177,156.992
C06186=1040.259,-10.219,418.809,169.280,37.176,156.992
C06187=1040.253,-10.468,418.824,169.278,37.176,156.992
C06188=1040.246,-10.718,418.837,169.275,37.175,156.992
C06189=1040.240,-10.967,418.852,169.273,37.174,156.992
C06190=1040.234,-11.217,418.867,169.271,37.174,156.992
C06191=1040.227,-11.467,418.880,169.269,37.173,156.991
C06192=1040.221,-11.716,418.895,169.267,37.172,156.991
C06193=1040.215,-11.965,418.910,169.265,37.172,156.991
C06194=1040.208,-12.215,418.924,169.263,37.171,156.991
C06195=1040.202,-12.464,418.938,169.261,37.171,156.991
C06196=1040.196,-12.714,418.953,169.259,37.170,156.991
C06197=1040.190,-12.963,418.966,169.256,37.169,156.991
C06198=1040.183,-13.213,418.981,169.254,37.169,156.990
C06199=1040.177,-13.463,418.996,169.252,37.168,156.990
C06200=1040.171,-13.712,419.010,169.250,37.168,156.990
C06201=1040.165,-13.962,419.024,169.248,37.167,156.990
C06202=1040.159,-14.211,419.038,169.246,37.166,156.990
C06203=1040.152,-14.460,419.053,169.244,37.166,156.990
C06204=1040.146,-14.710,419.067,169.242,37.165,156.990
C06205=1040.139,-14.959,419.081,169.240,37.165,156.990
C06206=1040.134,-15.209,419.095,169.237,37.164,156.989
C06207=1040.127,-15.459,419.110,169.235,37.164,156.989
C06208=1040.120,-15.708,419.123,169.233,37.163,156.989
C06209=1040.114,-15.957,419.137,169.230,37.163,156.989
C06210=1040.108,-16.207,419.152,169.228,37.162,156.989
C06211=1040.102,-16.457,419.165,169.226,37.162,156.989
C06212=1040.095,-16.706,419.180,169.224,37.161,156.989
C06213=1040.088,-16.956,419.193,169.222,37.161,156.989
C06214=1040.083,-17.205,419.208,169.220,37.160,156.989
C06215=1040.076,-17.455,419.222,169.218,37.160,156.989
C06216=1040.069,-17.704,419.236,169.215,37.159,156.988
C06217=1040.063,-17.954,419.250,169.213,37.159,156.988
C06218=1040.057,-18.203,419.263,169.211,37.158,156.988
C06219=1040.051,-18.453,419.278,169.209,37.158,156.988
C06220=1040.044,-18.702,419.291,169.207,37.157,156.988
C06221=1040.038,-18.952,419.305,169.205,37.157,156.988
C06222=1040.030,-19.234,419.321,169.202,37.156,156.988
C06223=1040.023,-19.515,419.337,169.199,37.156,156.988
C06224=1040.017,-19.798,419.353,169.197,37.155,156.988
C06225=1040.009,-20.080,419.369,169.194,37.154,156.987
C06226=1040.003,-20.329,419.382,169.192,37.154,156.987
C06227=1039.996,-20.578,419.397,169.190,37.153,156.987
C06228=1039.990,-20.828,419.410,169.188,37.153,156.987
C06229=1039.984,-21.078,419.424,169.186,37.153,156.987
C06230=1039.977,-21.327,419.437,169.184,37.152,156.987
C06231=1039.972,-21.576,419.452,169.182,37.151,156.987
C06232=1039.965,-21.826,419.466,169.179,37.151,156.987
C06233=1039.959,-22.076,419.479,169.177,37.150,156.987
C06234=1039.952,-22.325,419.494,169.175,37.150,156.987
C06235=1039.946,-22.574,419.507,169.173,37.150,156.986
C06236=1039.940,-22.825,419.521,169.170,37.149,156.986
C06237=1039.934,-23.074,419.535,169.168,37.148,156.986
C06238=1039.927,-23.324,419.548,169.166,37.148,156.986
C06239=1039.921,-23.573,419.563,169.164,37.148,156.986
C06240=1039.915,-23.822,419.576,169.161,37.147,156.986
C06241=1039.909,-24.072,419.590,169.159,37.147,156.986
C06242=1039.903,-24.322,419.604,169.157,37.146,156.986
C06243=1039.896,-24.572,419.617,169.155,37.145,156.986
C06244=1039.890,-24.821,419.632,169.153,37.145,156.985
C06245=1039.883,-25.070,419.645,169.151,37.145,156.985
C06246=1039.877,-25.320,419.659,169.149,37.144,156.985
C06247=1039.871,-25.569,419.673,169.146,37.144,156.985
C06248=1039.865,-25.819,419.686,169.144,37.143,156.985
C06249=1039.858,-26.069,419.699,169.142,37.142,156.985
C06250=1039.853,-26.317,419.714,169.139,37.142,156.985
C06251=1039.846,-26.567,419.728,169.137,37.142,156.985
C06252=1039.840,-26.817,419.741,169.135,37.141,156.985
C06253=1039.833,-27.067,419.755,169.133,37.141,156.985
C06254=1039.827,-27.316,419.768,169.130,37.140,156.984
C06255=1039.821,-27.566,419.782,169.128,37.140,156.984
C06256=1039.814,-27.815,419.795,169.126,37.139,156.984
C06257=1039.808,-28.065,419.809,169.124,37.139,156.984
C06258=1039.801,-28.315,419.822,169.122,37.139,156.984
C06259=1039.795,-28.564,419.835,169.120,37.138,156.984
C06260=1039.789,-28.813,419.849,169.117,37.138,156.984
C06261=1039.783,-29.064,419.863,169.115,37.138,156.984
C06262=1039.777,-29.313,419.876,169.113,37.137,156.984
C06263=1039.770,-29.562,419.890,169.111,37.136,156.984
C06264=1039.763,-29.812,419.903,169.109,37.136,156.984
C06265=1039.757,-30.061,419.916,169.106,37.136,156.983
C06266=1039.750,-30.311,419.930,169.103,37.135,156.983
C06267=1039.744,-30.561,419.943,169.101,37.135,156.983
C06268=1039.738,-30.810,419.957,169.099,37.135,156.983
C06269=1039.731,-31.060,419.970,169.097,37.134,156.983
C06270=1039.725,-31.309,419.984,169.094,37.134,156.983
C06271=1039.719,-31.558,419.997,169.092,37.133,156.983
C06272=1039.713,-31.808,420.009,169.090,37.133,156.983
C06273=1039.707,-32.058,420.024,169.088,37.133,156.983
C06274=1039.701,-32.308,420.037,169.086,37.132,156.983
C06275=1039.694,-32.557,420.050,169.083,37.132,156.983
C06276=1039.688,-32.807,420.064,169.081,37.132,156.983
C06277=1039.681,-33.056,420.077,169.079,37.131,156.982
C06278=1039.675,-33.305,420.090,169.077,37.130,156.982
C06279=1039.668,-33.555,420.104,169.075,37.131,156.982
C06280=1039.662,-33.805,420.116,169.072,37.130,156.982
C06281=1039.656,-34.055,420.130,169.070,37.129,156.982
C06282=1039.650,-34.304,420.143,169.068,37.129,156.982
C06283=1039.643,-34.554,420.157,169.065,37.129,156.982
C06284=1039.637,-34.803,420.170,169.063,37.129,156.982
C06285=1039.631,-35.053,420.182,169.060,37.128,156.982
C06286=1039.624,-35.334,420.198,169.058,37.128,156.982
C06287=1039.617,-35.615,420.213,169.055,37.127,156.982
C06288=1039.610,-35.896,420.228,169.053,37.127,156.982
C06289=1039.603,-36.177,420.242,169.050,37.126,156.981
C06290=1039.597,-36.427,420.256,169.048,37.126,156.981
C06291=1039.591,-36.676,420.269,169.046,37.126,156.981
C06292=1039.584,-36.926,420.283,169.044,37.125,156.981
C06293=1039.578,-37.176,420.295,169.042,37.125,156.981
C06294=1039.572,-37.425,420.308,169.039,37.125,156.981
C06295=1039.565,-37.674,420.322,169.037,37.124,156.981
C06296=1039.560,-37.924,420.334,169.035,37.123,156.981
C06297=1039.553,-38.173,420.348,169.033,37.123,156.981
C06298=1039.547,-38.423,420.361,169.031,37.123,156.981
C06299=1039.541,-38.673,420.374,169.028,37.123,156.981
C06300=1039.534,-38.922,420.387,169.026,37.122,156.981
C06301=1039.528,-39.172,420.400,169.023,37.122,156.980
C06302=1039.522,-39.422,420.413,169.021,37.122,156.980
C06303=1039.515,-39.672,420.426,169.018,37.121,156.980
C06304=1039.509,-39.921,420.439,169.016,37.121,156.980
C06305=1039.503,-40.170,420.452,169.014,37.121,156.980
C06306=1039.496,-40.420,420.465,169.011,37.121,156.980
C06307=1039.490,-40.670,420.478,169.009,37.121,156.980
C06308=1039.484,-40.920,420.491,169.007,37.120,156.980
C06309=1039.477,-41.169,420.503,169.005,37.120,156.980
C06310=1039.471,-41.418,420.516,169.002,37.119,156.980
C06311=1039.465,-41.668,420.530,169.000,37.119,156.980
C06312=1039.459,-41.917,420.542,168.998,37.119,156.980
C06313=1039.452,-42.167,420.555,168.996,37.119,156.980
C06314=1039.446,-42.416,420.567,168.993,37.118,156.980
C06315=1039.439,-42.666,420.581,168.991,37.118,156.980
C06316=1039.433,-42.916,420.594,168.989,37.118,156.979
C06317=1039.427,-43.165,420.607,168.987,37.118,156.979
C06318=1039.420,-43.415,420.619,168.984,37.117,156.979
C06319=1039.414,-43.664,420.632,168.982,37.117,156.979
C06320=1039.408,-43.914,420.645,168.980,37.117,156.979
C06321=1039.402,-44.164,420.657,168.977,37.117,156.979
C06322=1039.395,-44.413,420.670,168.975,37.116,156.979
C06323=1039.389,-44.663,420.682,168.973,37.116,156.979
C06324=1039.383,-44.913,420.696,168.971,37.116,156.979
C06325=1039.377,-45.163,420.709,168.967,37.115,156.979
C06326=1039.370,-45.412,420.722,168.965,37.115,156.979
C06327=1039.364,-45.662,420.734,168.963,37.115,156.979
C06328=1039.358,-45.911,420.746,168.960,37.115,156.979
C06329=1039.352,-46.161,420.760,168.958,37.114,156.979
C06330=1039.346,-46.411,420.772,168.956,37.114,156.979
C06331=1039.339,-46.660,420.785,168.954,37.114,156.978
C06332=1039.333,-46.909,420.797,168.951,37.114,156.978
C06333=1039.327,-47.159,420.810,168.949,37.113,156.978
C06334=1039.320,-47.408,420.823,168.947,37.113,156.978
C06335=1039.314,-47.658,420.835,168.944,37.113,156.978
C06336=1039.308,-47.908,420.848,168.942,37.113,156.978
C06337=1039.302,-48.157,420.861,168.940,37.113,156.978
C06338=1039.295,-48.407,420.873,168.938,37.112,156.978
C06339=1039.289,-48.657,420.886,168.935,37.112,156.978
C06340=1039.283,-48.906,420.899,168.933,37.111,156.978
C06341=1039.277,-49.156,420.911,168.931,37.111,156.978
C06342=1039.271,-49.405,420.923,168.928,37.111,156.978
C06343=1039.264,-49.655,420.937,168.926,37.111,156.978
C06344=1039.259,-49.905,420.949,168.924,37.110,156.978
C06345=1039.252,-50.154,420.961,168.921,37.110,156.978
C06346=1039.246,-50.404,420.974,168.919,37.110,156.978
C06347=1039.240,-50.653,420.987,168.917,37.110,156.978
C06348=1039.233,-50.903,420.999,168.914,37.110,156.978
C06349=1039.227,-51.153,421.011,168.912,37.110,156.978
C06350=1039.219,-51.435,421.025,168.909,37.110,156.978
C06351=1039.212,-51.716,421.039,168.906,37.109,156.977
C06352=1039.206,-51.997,421.052,168.903,37.109,156.977
C06353=1039.198,-52.279,421.067,168.900,37.109,156.977
C06354=1039.192,-52.528,421.079,168.898,37.109,156.977
C06355=1039.185,-52.778,421.091,168.896,37.109,156.977
C06356=1039.179,-53.028,421.103,168.893,37.109,156.977
C06357=1039.172,-53.277,421.115,168.891,37.109,156.977
C06358=1039.167,-53.527,421.128,168.889,37.109,156.977
C06359=1039.160,-53.777,421.140,168.886,37.109,156.977
C06360=1039.153,-54.026,421.152,168.884,37.109,156.977
C06361=1039.147,-54.276,421.164,168.882,37.108,156.977
C06362=1039.140,-54.525,421.177,168.879,37.108,156.977
C06363=1039.134,-54.775,421.189,168.877,37.108,156.977
C06364=1039.128,-55.025,421.201,168.874,37.108,156.977
C06365=1039.121,-55.274,421.213,168.872,37.108,156.977
C06366=1039.115,-55.524,421.225,168.870,37.108,156.977
C06367=1039.109,-55.774,421.238,168.867,37.108,156.977
C06368=1039.103,-56.023,421.250,168.865,37.108,156.977
C06369=1039.097,-56.272,421.262,168.863,37.108,156.977
C06370=1039.090,-56.522,421.274,168.860,37.108,156.977
C06371=1039.083,-56.772,421.286,168.858,37.108,156.977
C06372=1039.077,-57.021,421.299,168.855,37.107,156.977
C06373=1039.071,-57.271,421.311,168.853,37.107,156.977
C06374=1039.064,-57.521,421.322,168.851,37.107,156.977
C06375=1039.059,-57.771,421.334,168.848,37.108,156.977
C06376=1039.052,-58.021,421.346,168.846,37.108,156.977
C06377=1039.046,-58.270,421.358,168.843,37.108,156.977
C06378=1039.040,-58.519,421.370,168.841,37.107,156.977
C06379=1039.033,-58.769,421.382,168.839,37.107,156.977
C06380=1039.027,-59.019,421.394,168.836,37.107,156.977
C06381=1039.021,-59.268,421.407,168.834,37.107,156.977
C06382=1039.014,-59.518,421.419,168.832,37.107,156.977
C06383=1039.007,-59.768,421.431,168.829,37.107,156.977
C06384=1039.001,-60.016,421.442,168.827,37.107,156.976
C06385=1038.996,-60.267,421.454,168.824,37.107,156.976
C06386=1038.989,-60.517,421.466,168.822,37.107,156.976
C06387=1038.983,-60.766,421.478,168.820,37.107,156.976
C06388=1038.977,-61.016,421.491,168.817,37.107,156.976
C06389=1038.971,-61.265,421.502,168.815,37.107,156.976
C06390=1038.964,-61.514,421.514,168.812,37.107,156.976
C06391=1038.958,-61.765,421.526,168.810,37.107,156.976
C06392=1038.952,-62.014,421.538,168.808,37.106,156.976
C06393=1038.945,-62.264,421.550,168.805,37.106,156.976
C06394=1038.940,-62.513,421.562,168.803,37.106,156.976
C06395=1038.933,-62.763,421.574,168.800,37.106,156.976
C06396=1038.927,-63.013,421.585,168.798,37.106,156.976
C06397=1038.920,-63.263,421.597,168.796,37.106,156.976
C06398=1038.915,-63.512,421.610,168.793,37.106,156.976
C06399=1038.908,-63.761,421.622,168.791,37.106,156.976
C06400=1038.902,-64.012,421.633,168.788,37.106,156.976
C06401=1038.896,-64.261,421.645,168.786,37.106,156.976
C06402=1038.890,-64.510,421.657,168.784,37.106,156.976
C06403=1038.883,-64.760,421.669,168.781,37.106,156.976
C06404=1038.877,-65.010,421.680,168.778,37.106,156.976
C06405=1038.872,-65.259,421.692,168.775,37.106,156.976
C06406=1038.865,-65.509,421.704,168.773,37.106,156.976
C06407=1038.859,-65.759,421.715,168.771,37.106,156.976
C06408=1038.852,-66.009,421.727,168.768,37.106,156.976
C06409=1038.847,-66.258,421.740,168.766,37.106,156.976
C06410=1038.840,-66.508,421.751,168.763,37.106,156.976
C06411=1038.834,-66.758,421.763,168.761,37.106,156.976
C06412=1038.828,-67.006,421.774,168.758,37.106,156.976
C06413=1038.822,-67.257,421.786,168.756,37.106,156.976
C06414=1038.815,-67.540,421.799,168.753,37.106,156.976
C06415=1038.808,-67.822,421.813,168.751,37.106,156.976
C06416=1038.801,-68.105,421.826,168.748,37.106,156.976
C06417=1038.794,-68.388,421.839,168.745,37.105,156.976
C06418=1038.788,-68.638,421.851,168.743,37.105,156.976
C06419=1038.782,-68.887,421.862,168.740,37.105,156.976
C06420=1038.776,-69.137,421.875,168.738,37.105,156.976
C06421=1038.769,-69.387,421.886,168.735,37.105,156.976
C06422=1038.763,-69.636,421.898,168.733,37.105,156.976
C06423=1038.757,-69.886,421.909,168.731,37.105,156.976
C06424=1038.752,-70.135,421.921,168.728,37.106,156.976
C06425=1038.745,-70.385,421.932,168.726,37.106,156.976
C06426=1038.739,-70.635,421.944,168.723,37.106,156.976
C06427=1038.733,-70.884,421.955,168.721,37.106,156.976
C06428=1038.726,-71.134,421.967,168.718,37.106,156.976
C06429=1038.721,-71.384,421.979,168.716,37.105,156.975
C06430=1038.715,-71.633,421.990,168.714,37.105,156.975
C06431=1038.709,-71.883,422.001,168.711,37.105,156.975
C06432=1038.702,-72.132,422.013,168.709,37.105,156.975
C06433=1038.697,-72.383,422.025,168.706,37.105,156.975
C06434=1038.691,-72.632,422.037,168.704,37.105,156.975
C06435=1038.684,-72.882,422.048,168.701,37.105,156.975
C06436=1038.679,-73.131,422.059,168.699,37.105,156.975
C06437=1038.672,-73.381,422.071,168.696,37.105,156.975
C06438=1038.667,-73.631,422.082,168.694,37.105,156.975
C06439=1038.660,-73.880,422.094,168.692,37.105,156.975
C06440=1038.655,-74.130,422.105,168.689,37.105,156.975
C06441=1038.648,-74.380,422.116,168.687,37.106,156.975
C06442=1038.642,-74.629,422.128,168.684,37.106,156.975
C06443=1038.636,-74.879,422.139,168.682,37.106,156.975
C06444=1038.630,-75.129,422.150,168.679,37.106,156.975
C06445=1038.623,-75.378,422.162,168.677,37.106,156.975
C06446=1038.617,-75.628,422.173,168.674,37.106,156.975
C06447=1038.611,-75.878,422.184,168.672,37.106,156.975
C06448=1038.605,-76.128,422.195,168.669,37.106,156.975
C06449=1038.598,-76.377,422.206,168.667,37.106,156.975
C06450=1038.592,-76.627,422.218,168.664,37.107,156.975
C06451=1038.586,-76.876,422.229,168.662,37.107,156.975
C06452=1038.580,-77.126,422.240,168.659,37.107,156.975
C06453=1038.574,-77.375,422.251,168.657,37.107,156.975
C06454=1038.567,-77.625,422.263,168.654,37.107,156.975
C06455=1038.562,-77.875,422.273,168.652,37.107,156.975
C06456=1038.555,-78.125,422.285,168.649,37.107,156.975
C06457=1038.549,-78.374,422.296,168.647,37.107,156.975
C06458=1038.543,-78.624,422.308,168.644,37.108,156.975
C06459=1038.537,-78.874,422.318,168.642,37.108,156.975
C06460=1038.532,-79.123,422.329,168.639,37.108,156.975
C06461=1038.525,-79.373,422.341,168.637,37.108,156.975
C06462=1038.519,-79.623,422.351,168.634,37.108,156.975
C06463=1038.512,-79.872,422.363,168.632,37.108,156.975
C06464=1038.506,-80.122,422.374,168.629,37.109,156.975
C06465=1038.500,-80.372,422.385,168.627,37.109,156.975
C06466=1038.494,-80.621,422.396,168.624,37.109,156.975
C06467=1038.487,-80.871,422.406,168.622,37.110,156.976
C06468=1038.481,-81.121,422.417,168.619,37.110,156.976
C06469=1038.475,-81.371,422.429,168.617,37.111,156.976
C06470=1038.469,-81.620,422.439,168.614,37.111,156.976
C06471=1038.462,-81.870,422.450,168.612,37.111,156.976
C06472=1038.457,-82.120,422.461,168.609,37.111,156.976
C06473=1038.450,-82.369,422.471,168.606,37.111,156.976
C06474=1038.444,-82.619,422.483,168.604,37.111,156.976
C06475=1038.438,-82.869,422.493,168.601,37.112,156.976
C06476=1038.431,-83.118,422.504,168.599,37.112,156.976
C06477=1038.425,-83.368,422.515,168.596,37.112,156.976
C06478=1038.418,-83.653,422.527,168.594,37.113,156.976
C06479=1038.411,-83.937,422.540,168.591,37.113,156.976
C06480=1038.403,-84.223,422.552,168.589,37.114,156.976
C06481=1038.396,-84.508,422.564,168.586,37.114,156.976
C06482=1038.390,-84.758,422.575,168.583,37.114,156.976
C06483=1038.385,-85.007,422.586,168.581,37.114,156.976
C06484=1038.378,-85.257,422.597,168.578,37.114,156.976
C06485=1038.372,-85.506,422.608,168.575,37.115,156.976
C06486=1038.365,-85.756,422.618,168.573,37.115,156.976
C06487=1038.359,-86.006,422.629,168.570,37.115,156.976
C06488=1038.354,-86.256,422.639,168.568,37.116,156.976
C06489=1038.347,-86.506,422.650,168.565,37.116,156.976
C06490=1038.341,-86.755,422.661,168.563,37.117,156.976
C06491=1038.335,-87.005,422.672,168.560,37.117,156.976
C06492=1038.328,-87.255,422.682,168.558,37.117,156.976
C06493=1038.322,-87.504,422.693,168.555,37.117,156.976
C06494=1038.317,-87.754,422.704,168.552,37.117,156.976
C06495=1038.310,-88.003,422.714,168.550,37.118,156.977
C06496=1038.304,-88.254,422.725,168.547,37.118,156.977
C06497=1038.297,-88.503,422.735,168.545,37.119,156.977
C06498=1038.292,-88.752,422.746,168.542,37.119,156.977
C06499=1038.285,-89.002,422.757,168.540,37.119,156.977
C06500=1038.279,-89.252,422.767,168.537,37.120,156.977
C06501=1038.273,-89.502,422.778,168.535,37.120,156.977
C06502=1038.267,-89.751,422.788,168.532,37.120,156.977
C06503=1038.261,-90.001,422.799,168.529,37.120,156.977
C06504=1038.255,-90.251,422.810,168.527,37.121,156.977
C06505=1038.249,-90.500,422.820,168.524,37.121,156.977
C06506=1038.243,-90.750,422.831,168.522,37.121,156.977
C06507=1038.237,-91.000,422.842,168.519,37.122,156.977
C06508=1038.231,-91.250,422.852,168.517,37.122,156.977
C06509=1038.225,-91.499,422.862,168.514,37.123,156.977
C06510=1038.218,-91.749,422.873,168.511,37.123,156.977
C06511=1038.212,-91.999,422.883,168.509,37.123,156.977
C06512=1038.206,-92.249,422.894,168.506,37.123,156.977
C06513=1038.200,-92.498,422.904,168.505,37.124,156.977
C06514=1038.194,-92.747,422.915,168.502,37.124,156.977
C06515=1038.188,-92.997,422.925,168.500,37.125,156.977
C06516=1038.182,-93.247,422.936,168.497,37.125,156.977
C06517=1038.176,-93.497,422.946,168.494,37.126,156.977
C06518=1038.170,-93.747,422.957,168.492,37.126,156.977
C06519=1038.164,-93.996,422.967,168.489,37.126,156.977
C06520=1038.158,-94.246,422.977,168.487,37.126,156.978
C06521=1038.152,-94.496,422.988,168.484,37.126,156.978
C06522=1038.145,-94.745,422.999,168.482,37.127,156.978
C06523=1038.140,-94.996,423.009,168.479,37.127,156.978
C06524=1038.133,-95.245,423.019,168.476,37.128,156.978
C06525=1038.128,-95.495,423.029,168.474,37.128,156.978
C06526=1038.121,-95.744,423.039,168.471,37.129,156.978
C06527=1038.116,-95.993,423.050,168.469,37.129,156.978
C06528=1038.110,-96.244,423.060,168.466,37.129,156.978
C06529=1038.104,-96.493,423.071,168.463,37.129,156.978
C06530=1038.098,-96.744,423.081,168.461,37.130,156.978
C06531=1038.091,-96.993,423.092,168.458,37.130,156.978
C06532=1038.086,-97.243,423.102,168.456,37.131,156.978
C06533=1038.079,-97.492,423.112,168.453,37.131,156.978
C06534=1038.074,-97.742,423.122,168.451,37.132,156.978
C06535=1038.067,-97.991,423.132,168.448,37.132,156.978
C06536=1038.061,-98.241,423.142,168.445,37.133,156.978
C06537=1038.056,-98.491,423.152,168.443,37.133,156.978
C06538=1038.049,-98.740,423.162,168.440,37.134,156.978
C06539=1038.042,-98.991,423.172,168.437,37.134,156.979
C06540=1038.037,-99.240,423.183,168.435,37.134,156.979
C06541=1038.031,-99.490,423.193,168.433,37.135,156.979
C06542=1038.023,-99.778,423.204,168.430,37.136,156.979
C06543=1038.017,-100.064,423.216,168.427,37.137,156.979
C06544=1038.010,-100.351,423.227,168.424,37.137,156.979
C06545=1038.002,-100.638,423.239,168.421,37.137,156.979
C06546=1037.997,-100.889,423.249,168.418,37.138,156.979
C06547=1037.990,-101.138,423.259,168.416,37.139,156.979
C06548=1037.984,-101.388,423.269,168.413,37.139,156.979
C06549=1037.978,-101.637,423.278,168.411,37.140,156.979
C06550=1037.972,-101.887,423.289,168.408,37.140,156.979
C06551=1037.966,-102.137,423.299,168.405,37.141,156.979
C06552=1037.959,-102.387,423.309,168.403,37.141,156.979
C06553=1037.954,-102.637,423.320,168.400,37.142,156.980
C06554=1037.948,-102.886,423.329,168.397,37.142,156.980
C06555=1037.941,-103.136,423.339,168.395,37.143,156.980
C06556=1037.935,-103.386,423.348,168.392,37.143,156.980
C06557=1037.929,-103.636,423.359,168.390,37.144,156.980
C06558=1037.923,-103.885,423.369,168.387,37.145,156.980
C06559=1037.917,-104.135,423.378,168.385,37.145,156.980
C06560=1037.911,-104.385,423.388,168.383,37.145,156.980
C06561=1037.905,-104.634,423.399,168.380,37.146,156.980
C06562=1037.899,-104.884,423.408,168.377,37.147,156.980
C06563=1037.893,-105.134,423.418,168.375,37.147,156.980
C06564=1037.887,-105.383,423.427,168.372,37.148,156.980
C06565=1037.882,-105.633,423.437,168.369,37.148,156.980
C06566=1037.876,-105.883,423.447,168.367,37.149,156.981
C06567=1037.869,-106.132,423.457,168.364,37.150,156.981
C06568=1037.863,-106.382,423.467,168.361,37.150,156.981
C06569=1037.857,-106.632,423.476,168.359,37.151,156.981
C06570=1037.851,-106.882,423.486,168.356,37.151,156.981
C06571=1037.845,-107.132,423.496,168.353,37.152,156.981
C06572=1037.839,-107.381,423.505,168.351,37.152,156.981
C06573=1037.833,-107.631,423.515,168.348,37.153,156.981
C06574=1037.827,-107.881,423.525,168.346,37.154,156.981
C06575=1037.820,-108.130,423.535,168.343,37.154,156.981
C06576=1037.814,-108.380,423.544,168.341,37.155,156.981
C06577=1037.808,-108.630,423.554,168.338,37.156,156.982
C06578=1037.802,-108.880,423.564,168.336,37.157,156.982
C06579=1037.796,-109.130,423.574,168.333,37.157,156.982
C06580=1037.790,-109.380,423.583,168.330,37.158,156.982
C06581=1037.785,-109.629,423.593,168.328,37.158,156.982
C06582=1037.778,-109.878,423.602,168.325,37.159,156.982
C06583=1037.772,-110.128,423.612,168.322,37.159,156.982
C06584=1037.766,-110.378,423.621,168.320,37.160,156.982
C06585=1037.760,-110.628,423.631,168.317,37.161,156.982
C06586=1037.754,-110.878,423.640,168.314,37.162,156.982
C06587=1037.748,-111.127,423.650,168.312,37.162,156.982
C06588=1037.741,-111.377,423.659,168.309,37.163,156.983
C06589=1037.736,-111.626,423.669,168.306,37.164,156.983
C06590=1037.730,-111.876,423.678,168.304,37.164,156.983
C06591=1037.724,-112.127,423.687,168.302,37.165,156.983
C06592=1037.718,-112.376,423.697,168.299,37.166,156.983
C06593=1037.711,-112.626,423.706,168.297,37.167,156.983
C06594=1037.705,-112.876,423.716,168.294,37.167,156.983
C06595=1037.699,-113.126,423.725,168.291,37.168,156.983
C06596=1037.693,-113.375,423.735,168.289,37.169,156.983
C06597=1037.687,-113.625,423.744,168.286,37.169,156.983
C06598=1037.681,-113.874,423.754,168.283,37.170,156.984
C06599=1037.675,-114.124,423.763,168.281,37.171,156.984
C06600=1037.669,-114.375,423.772,168.278,37.171,156.984
C06601=1037.664,-114.624,423.781,168.275,37.172,156.984
C06602=1037.657,-114.874,423.791,168.273,37.173,156.984
C06603=1037.651,-115.123,423.800,168.270,37.174,156.984
C06604=1037.645,-115.373,423.810,168.267,37.174,156.984
C06605=1037.639,-115.623,423.820,168.265,37.175,156.984
C06606=1037.633,-115.909,423.830,168.262,37.176,156.984
C06607=1037.625,-116.195,423.840,168.259,37.177,156.985
C06608=1037.619,-116.482,423.851,168.256,37.178,156.985
C06609=1037.612,-116.768,423.862,168.253,37.179,156.985
C06610=1037.605,-117.018,423.870,168.250,37.179,156.985
C06611=1037.599,-117.268,423.880,168.248,37.181,156.985
C06612=1037.594,-117.517,423.889,168.245,37.181,156.985
C06613=1037.587,-117.767,423.899,168.242,37.182,156.985
C06614=1037.581,-118.018,423.908,168.240,37.183,156.985
C06615=1037.575,-118.267,423.917,168.237,37.183,156.985
C06616=1037.570,-118.516,423.926,168.234,37.184,156.986
C06617=1037.564,-118.767,423.935,168.232,37.185,156.986
C06618=1037.557,-119.016,423.944,168.230,37.186,156.986
C06619=1037.551,-119.266,423.954,168.227,37.187,156.986
C06620=1037.546,-119.516,423.962,168.224,37.188,156.986
C06621=1037.539,-119.766,423.972,168.222,37.188,156.986
C06622=1037.533,-120.015,423.981,168.219,37.189,156.986
C06623=1037.528,-120.265,423.990,168.216,37.190,156.986
C06624=1037.521,-120.515,423.999,168.213,37.191,156.987
C06625=1037.515,-120.764,424.008,168.211,37.192,156.987
C06626=1037.510,-121.014,424.017,168.208,37.193,156.987
C06627=1037.503,-121.264,424.026,168.205,37.193,156.987
C06628=1037.498,-121.514,424.035,168.204,37.194,156.987
C06629=1037.491,-121.763,424.044,168.201,37.195,156.987
C06630=1037.485,-122.014,424.053,168.198,37.196,156.987
C06631=1037.479,-122.263,424.062,168.195,37.197,156.987
C06632=1037.474,-122.512,424.071,168.193,37.197,156.988
C06633=1037.468,-122.763,424.080,168.190,37.198,156.988
C06634=1037.461,-123.012,424.089,168.187,37.200,156.988
C06635=1037.456,-123.262,424.098,168.184,37.200,156.988
C06636=1037.449,-123.512,424.107,168.182,37.201,156.988
C06637=1037.444,-123.762,424.116,168.179,37.202,156.988
C06638=1037.438,-124.011,424.125,168.176,37.203,156.988
C06639=1037.431,-124.262,424.134,168.175,37.204,156.988
C06640=1037.426,-124.511,424.143,168.172,37.204,156.989
C06641=1037.420,-124.761,424.152,168.169,37.206,156.989
C06642=1037.413,-125.011,424.161,168.166,37.207,156.989
C06643=1037.408,-125.260,424.169,168.164,37.207,156.989
C06644=1037.402,-125.511,424.178,168.161,37.209,156.989
C06645=1037.396,-125.759,424.187,168.158,37.209,156.989
C06646=1037.390,-126.010,424.195,168.155,37.210,156.989
C06647=1037.384,-126.260,424.205,168.153,37.211,156.990
C06648=1037.378,-126.509,424.213,168.150,37.212,156.990
C06649=1037.372,-126.760,424.222,168.148,37.213,156.990
C06650=1037.366,-127.009,424.231,168.145,37.214,156.990
C06651=1037.360,-127.259,424.239,168.143,37.215,156.990
C06652=1037.354,-127.508,424.248,168.140,37.216,156.990
C06653=1037.347,-127.758,424.257,168.137,37.217,156.990
C06654=1037.342,-128.007,424.266,168.135,37.218,156.990
C06655=1037.338,-128.257,424.276,168.132,37.218,156.990
C06656=1037.333,-128.507,424.285,168.130,37.218,156.990
C06657=1037.330,-128.757,424.296,168.127,37.217,156.990
C06658=1037.327,-129.007,424.308,168.125,37.216,156.990
C06659=1037.326,-129.256,424.320,168.124,37.215,156.990
C06660=1037.325,-129.507,424.333,168.121,37.212,156.989
C06661=1037.324,-129.756,424.346,168.119,37.210,156.989
C06662=1037.325,-130.007,424.360,168.118,37.207,156.988
C06663=1037.326,-130.256,424.374,168.116,37.203,156.988
C06664=1037.327,-130.507,424.389,168.115,37.200,156.987
C06665=1037.331,-130.757,424.404,168.113,37.196,156.987
C06666=1037.334,-131.007,424.421,168.112,37.190,156.986
C06667=1037.339,-131.257,424.437,168.110,37.185,156.985
C06668=1037.343,-131.508,424.455,168.109,37.180,156.984
C06669=1037.350,-131.757,424.473,168.109,37.174,156.983
C06670=1037.010,-131.781,424.201,168.061,37.382,157.017
C06671=1037.005,-131.532,424.184,168.061,37.388,157.018
C06672=1037.000,-131.282,424.166,168.062,37.394,157.019
C06673=1036.995,-131.032,424.149,168.064,37.399,157.020
C06674=1036.992,-130.781,424.133,168.065,37.404,157.021
C06675=1036.989,-130.531,424.118,168.067,37.408,157.022
C06676=1036.988,-130.281,424.102,168.068,37.411,157.022
C06677=1036.986,-130.031,424.088,168.070,37.415,157.023
C06678=1036.985,-129.781,424.075,168.071,37.418,157.024
C06679=1036.985,-129.531,424.061,168.074,37.421,157.024
C06680=1036.986,-129.281,424.048,168.075,37.423,157.024
C06681=1036.988,-129.032,424.037,168.077,37.424,157.025
C06682=1036.991,-128.781,424.025,168.079,37.425,157.025
C06683=1036.994,-128.531,424.014,168.082,37.426,157.025
C06684=1036.998,-128.281,424.004,168.084,37.426,157.025
C06685=1037.003,-128.032,423.994,168.086,37.426,157.025
C06686=1037.008,-127.783,423.984,168.089,37.425,157.025
C06687=1037.014,-127.533,423.976,168.092,37.424,157.025
C06688=1037.020,-127.283,423.968,168.095,37.423,157.025
C06689=1037.026,-127.034,423.959,168.097,37.422,157.025
C06690=1037.032,-126.784,423.950,168.100,37.421,157.024
C06691=1037.038,-126.533,423.941,168.103,37.420,157.024
C06692=1037.044,-126.284,423.933,168.106,37.419,157.024
C06693=1037.050,-126.034,423.924,168.107,37.419,157.024
C06694=1037.056,-125.785,423.915,168.110,37.417,157.024
C06695=1037.062,-125.535,423.906,168.113,37.416,157.024
C06696=1037.068,-125.284,423.898,168.116,37.415,157.024
C06697=1037.074,-125.035,423.888,168.118,37.414,157.023
C06698=1037.080,-124.785,423.880,168.121,37.414,157.023
C06699=1037.086,-124.536,423.871,168.124,37.412,157.023
C06700=1037.092,-124.286,423.862,168.127,37.411,157.023
C06701=1037.099,-124.036,423.853,168.129,37.411,157.023
C06702=1037.104,-123.786,423.845,168.131,37.409,157.023
C06703=1037.110,-123.537,423.835,168.134,37.409,157.023
C06704=1037.115,-123.287,423.826,168.137,37.408,157.023
C06705=1037.122,-123.037,423.817,168.139,37.406,157.022
C06706=1037.128,-122.787,423.809,168.142,37.406,157.022
C06707=1037.134,-122.538,423.799,168.145,37.405,157.022
C06708=1037.140,-122.288,423.791,168.148,37.404,157.022
C06709=1037.146,-122.038,423.781,168.150,37.403,157.022
C06710=1037.152,-121.788,423.773,168.153,37.402,157.022
C06711=1037.158,-121.539,423.764,168.156,37.401,157.022
C06712=1037.164,-121.288,423.755,168.159,37.401,157.022
C06713=1037.169,-121.039,423.746,168.160,37.399,157.021
C06714=1037.176,-120.789,423.736,168.163,37.399,157.021
C06715=1037.182,-120.539,423.728,168.166,37.398,157.021
C06716=1037.188,-120.290,423.719,168.168,37.397,157.021
C06717=1037.194,-120.040,423.709,168.171,37.396,157.021
C06718=1037.200,-119.790,423.700,168.174,37.395,157.021
C06719=1037.205,-119.541,423.691,168.177,37.394,157.021
C06720=1037.211,-119.290,423.682,168.179,37.394,157.021
C06721=1037.218,-119.041,423.673,168.182,37.393,157.020
C06722=1037.224,-118.791,423.664,168.185,37.391,157.020
C06723=1037.230,-118.541,423.655,168.187,37.391,157.020
C06724=1037.236,-118.292,423.645,168.189,37.390,157.020
C06725=1037.242,-118.042,423.636,168.192,37.389,157.020
C06726=1037.247,-117.792,423.627,168.195,37.389,157.020
C06727=1037.253,-117.542,423.618,168.198,37.387,157.020
C06728=1037.260,-117.293,423.609,168.200,37.386,157.020
C06729=1037.266,-117.043,423.599,168.203,37.386,157.019
C06730=1037.272,-116.793,423.591,168.206,37.385,157.019
C06731=1037.278,-116.507,423.580,168.209,37.384,157.019
C06732=1037.285,-116.220,423.569,168.212,37.383,157.019
C06733=1037.293,-115.934,423.559,168.215,37.382,157.019
C06734=1037.299,-115.647,423.548,168.218,37.381,157.019
C06735=1037.305,-115.397,423.538,168.220,37.381,157.019
C06736=1037.312,-115.147,423.529,168.223,37.380,157.019
C06737=1037.317,-114.898,423.520,168.225,37.379,157.018
C06738=1037.323,-114.649,423.510,168.228,37.378,157.018
C06739=1037.330,-114.398,423.502,168.231,37.377,157.018
C06740=1037.336,-114.149,423.492,168.233,37.376,157.018
C06741=1037.342,-113.899,423.483,168.236,37.376,157.018
C06742=1037.348,-113.650,423.473,168.239,37.375,157.018
C06743=1037.353,-113.400,423.463,168.242,37.374,157.018
C06744=1037.360,-113.150,423.454,168.244,37.374,157.018
C06745=1037.366,-112.900,423.444,168.247,37.373,157.018
C06746=1037.372,-112.650,423.435,168.250,37.372,157.018
C06747=1037.377,-112.401,423.426,168.251,37.371,157.017
C06748=1037.383,-112.151,423.417,168.254,37.371,157.017
C06749=1037.389,-111.901,423.407,168.257,37.370,157.017
C06750=1037.396,-111.651,423.397,168.259,37.369,157.017
C06751=1037.402,-111.401,423.388,168.262,37.368,157.017
C06752=1037.408,-111.152,423.378,168.265,37.368,157.017
C06753=1037.414,-110.902,423.369,168.268,37.367,157.017
C06754=1037.420,-110.653,423.359,168.270,37.366,157.017
C06755=1037.426,-110.403,423.350,168.273,37.366,157.017
C06756=1037.432,-110.153,423.340,168.276,37.365,157.017
C06757=1037.438,-109.903,423.331,168.278,37.364,157.017
C06758=1037.444,-109.654,423.321,168.281,37.363,157.016
C06759=1037.451,-109.404,423.312,168.284,37.363,157.016
C06760=1037.457,-109.154,423.302,168.285,37.362,157.016
C06761=1037.463,-108.904,423.293,168.288,37.361,157.016
C06762=1037.469,-108.654,423.283,168.291,37.361,157.016
C06763=1037.475,-108.405,423.274,168.293,37.360,157.016
C06764=1037.480,-108.155,423.264,168.296,37.359,157.016
C06765=1037.486,-107.905,423.254,168.299,37.358,157.016
C06766=1037.492,-107.656,423.244,168.302,37.358,157.016
C06767=1037.499,-107.406,423.235,168.304,37.357,157.016
C06768=1037.505,-107.156,423.225,168.307,37.356,157.015
C06769=1037.511,-106.907,423.215,168.310,37.356,157.015
C06770=1037.517,-106.657,423.205,168.312,37.355,157.015
C06771=1037.523,-106.407,423.195,168.315,37.355,157.015
C06772=1037.529,-106.157,423.186,168.318,37.354,157.015
C06773=1037.535,-105.907,423.176,168.320,37.353,157.015
C06774=1037.541,-105.657,423.167,168.323,37.353,157.015
C06775=1037.548,-105.408,423.157,168.325,37.352,157.015
C06776=1037.553,-105.158,423.146,168.327,37.351,157.015
C06777=1037.559,-104.908,423.137,168.330,37.350,157.015
C06778=1037.566,-104.659,423.127,168.333,37.350,157.015
C06779=1037.572,-104.409,423.117,168.335,37.350,157.015
C06780=1037.577,-104.159,423.107,168.338,37.349,157.014
C06781=1037.584,-103.909,423.097,168.340,37.348,157.014
C06782=1037.590,-103.660,423.087,168.343,37.348,157.014
C06783=1037.596,-103.410,423.078,168.346,37.347,157.014
C06784=1037.601,-103.160,423.068,168.348,37.347,157.014
C06785=1037.608,-102.911,423.057,168.351,37.346,157.014
C06786=1037.614,-102.661,423.048,168.354,37.345,157.014
C06787=1037.620,-102.411,423.038,168.356,37.345,157.014
C06788=1037.626,-102.161,423.028,168.359,37.345,157.014
C06789=1037.632,-101.912,423.018,168.362,37.344,157.014
C06790=1037.638,-101.662,423.008,168.364,37.343,157.014
C06791=1037.644,-101.412,422.998,168.367,37.342,157.014
C06792=1037.650,-101.163,422.988,168.370,37.342,157.014
C06793=1037.656,-100.913,422.978,168.371,37.342,157.014
C06794=1037.663,-100.663,422.969,168.374,37.341,157.013
C06795=1037.670,-100.376,422.956,168.377,37.340,157.013
C06796=1037.677,-100.089,422.945,168.380,37.339,157.013
C06797=1037.684,-99.801,422.934,168.383,37.339,157.013
C06798=1037.690,-99.514,422.922,168.386,37.338,157.013
C06799=1037.697,-99.265,422.912,168.389,37.338,157.013
C06800=1037.703,-99.015,422.902,168.391,37.337,157.013
C06801=1037.709,-98.765,422.892,168.394,37.336,157.013
C06802=1037.715,-98.515,422.882,168.397,37.336,157.013
C06803=1037.721,-98.266,422.872,168.399,37.336,157.013
C06804=1037.727,-98.016,422.861,168.402,37.335,157.013
C06805=1037.733,-97.766,422.852,168.405,37.334,157.013
C06806=1037.740,-97.517,422.841,168.407,37.334,157.013
C06807=1037.745,-97.267,422.831,168.410,37.334,157.013
C06808=1037.752,-97.018,422.821,168.412,37.333,157.012
C06809=1037.758,-96.767,422.810,168.415,37.333,157.012
C06810=1037.764,-96.518,422.800,168.418,37.332,157.012
C06811=1037.770,-96.268,422.790,168.420,37.332,157.012
C06812=1037.775,-96.018,422.779,168.422,37.331,157.012
C06813=1037.782,-95.769,422.769,168.424,37.331,157.012
C06814=1037.787,-95.519,422.759,168.427,37.330,157.012
C06815=1037.794,-95.269,422.749,168.430,37.330,157.012
C06816=1037.799,-95.020,422.738,168.432,37.330,157.012
C06817=1037.806,-94.770,422.727,168.435,37.329,157.012
C06818=1037.812,-94.520,422.717,168.437,37.329,157.012
C06819=1037.817,-94.270,422.706,168.440,37.328,157.012
C06820=1037.824,-94.020,422.697,168.443,37.328,157.012
C06821=1037.829,-93.771,422.686,168.445,37.327,157.012
C06822=1037.836,-93.522,422.676,168.448,37.327,157.012
C06823=1037.841,-93.272,422.666,168.450,37.327,157.012
C06824=1037.848,-93.022,422.655,168.453,37.327,157.012
C06825=1037.854,-92.772,422.644,168.456,37.326,157.012
C06826=1037.860,-92.522,422.634,168.458,37.326,157.012
C06827=1037.866,-92.273,422.624,168.461,37.325,157.012
C06828=1037.872,-92.024,422.613,168.463,37.325,157.012
C06829=1037.879,-91.773,422.603,168.466,37.324,157.011
C06830=1037.884,-91.524,422.592,168.469,37.324,157.011
C06831=1037.890,-91.274,422.581,168.471,37.324,157.011
C06832=1037.896,-91.024,422.571,168.474,37.324,157.011
C06833=1037.903,-90.774,422.560,168.476,37.323,157.011
C06834=1037.909,-90.525,422.550,168.479,37.323,157.011
C06835=1037.915,-90.275,422.539,168.481,37.322,157.011
C06836=1037.920,-90.025,422.529,168.484,37.322,157.011
C06837=1037.927,-89.776,422.519,168.487,37.321,157.011
C06838=1037.933,-89.526,422.507,168.489,37.321,157.011
C06839=1037.940,-89.277,422.497,168.492,37.321,157.011
C06840=1037.945,-89.027,422.487,168.494,37.321,157.011
C06841=1037.951,-88.776,422.476,168.496,37.320,157.011
C06842=1037.958,-88.527,422.465,168.499,37.320,157.011
C06843=1037.963,-88.278,422.454,168.501,37.319,157.011
C06844=1037.970,-88.029,422.444,168.504,37.319,157.011
C06845=1037.976,-87.778,422.434,168.506,37.318,157.011
C06846=1037.982,-87.528,422.423,168.509,37.318,157.011
C06847=1037.988,-87.279,422.412,168.511,37.318,157.011
C06848=1037.995,-87.029,422.401,168.514,37.317,157.011
C06849=1038.000,-86.779,422.390,168.517,37.317,157.011
C06850=1038.007,-86.530,422.380,168.519,37.317,157.011
C06851=1038.013,-86.280,422.369,168.522,37.317,157.011
C06852=1038.019,-86.030,422.359,168.524,37.316,157.011
C06853=1038.025,-85.781,422.348,168.527,37.316,157.011
C06854=1038.031,-85.531,422.337,168.529,37.315,157.010
C06855=1038.038,-85.281,422.327,168.532,37.315,157.010
C06856=1038.044,-85.032,422.316,168.535,37.314,157.010
C06857=1038.050,-84.782,422.305,168.537,37.314,157.010
C06858=1038.056,-84.533,422.294,168.540,37.314,157.010
C06859=1038.064,-84.247,422.282,168.543,37.314,157.010
C06860=1038.070,-83.963,422.270,168.546,37.313,157.010
C06861=1038.077,-83.677,422.257,168.548,37.313,157.010
C06862=1038.085,-83.392,422.244,168.551,37.313,157.010
C06863=1038.091,-83.143,422.234,168.554,37.312,157.010
C06864=1038.097,-82.894,422.223,168.557,37.312,157.010
C06865=1038.103,-82.643,422.212,168.559,37.311,157.010
C06866=1038.110,-82.394,422.202,168.562,37.311,157.010
C06867=1038.116,-82.144,422.190,168.564,37.310,157.010
C06868=1038.122,-81.894,422.180,168.567,37.310,157.010
C06869=1038.129,-81.645,422.169,168.569,37.310,157.010
C06870=1038.135,-81.395,422.158,168.572,37.310,157.010
C06871=1038.140,-81.146,422.147,168.574,37.310,157.010
C06872=1038.147,-80.896,422.136,168.577,37.309,157.010
C06873=1038.153,-80.646,422.126,168.580,37.309,157.010
C06874=1038.160,-80.396,422.114,168.582,37.309,157.010
C06875=1038.166,-80.147,422.104,168.584,37.308,157.010
C06876=1038.172,-79.897,422.093,168.586,37.308,157.010
C06877=1038.178,-79.647,422.082,168.589,37.308,157.010
C06878=1038.184,-79.397,422.071,168.591,37.307,157.010
C06879=1038.190,-79.147,422.060,168.594,37.307,157.010
C06880=1038.197,-78.898,422.048,168.596,37.307,157.010
C06881=1038.203,-78.648,422.037,168.599,37.307,157.010
C06882=1038.209,-78.398,422.026,168.601,37.307,157.010
C06883=1038.215,-78.149,422.015,168.604,37.306,157.010
C06884=1038.222,-77.899,422.004,168.606,37.306,157.010
C06885=1038.228,-77.650,421.993,168.609,37.306,157.010
C06886=1038.233,-77.401,421.982,168.611,37.306,157.010
C06887=1038.240,-77.150,421.971,168.614,37.305,157.010
C06888=1038.246,-76.901,421.960,168.616,37.305,157.010
C06889=1038.252,-76.651,421.948,168.619,37.305,157.010
C06890=1038.258,-76.402,421.937,168.621,37.305,157.010
C06891=1038.264,-76.152,421.926,168.624,37.305,157.010
C06892=1038.271,-75.901,421.914,168.626,37.305,157.009
C06893=1038.277,-75.653,421.903,168.629,37.305,157.009
C06894=1038.283,-75.402,421.891,168.631,37.304,157.009
C06895=1038.289,-75.153,421.881,168.634,37.304,157.010
C06896=1038.295,-74.903,421.869,168.636,37.304,157.010
C06897=1038.301,-74.654,421.858,168.639,37.304,157.009
C06898=1038.307,-74.404,421.847,168.641,37.304,157.009
C06899=1038.314,-74.155,421.836,168.644,37.304,157.009
C06900=1038.320,-73.905,421.824,168.646,37.304,157.009
C06901=1038.326,-73.655,421.813,168.649,37.303,157.009
C06902=1038.332,-73.405,421.801,168.651,37.303,157.009
C06903=1038.338,-73.156,421.790,168.654,37.303,157.010
C06904=1038.344,-72.906,421.779,168.656,37.303,157.010
C06905=1038.350,-72.656,421.766,168.659,37.303,157.010
C06906=1038.356,-72.406,421.755,168.661,37.303,157.010
C06907=1038.363,-72.157,421.743,168.664,37.303,157.010
C06908=1038.368,-71.907,421.732,168.666,37.303,157.010
C06909=1038.375,-71.658,421.720,168.668,37.303,157.010
C06910=1038.380,-71.408,421.709,168.671,37.303,157.010
C06911=1038.387,-71.158,421.697,168.673,37.303,157.010
C06912=1038.392,-70.909,421.686,168.676,37.303,157.010
C06913=1038.399,-70.659,421.674,168.678,37.303,157.010
C06914=1038.405,-70.409,421.662,168.681,37.303,157.010
C06915=1038.411,-70.160,421.651,168.683,37.303,157.010
C06916=1038.417,-69.910,421.640,168.686,37.303,157.010
C06917=1038.423,-69.661,421.628,168.688,37.303,157.010
C06918=1038.429,-69.410,421.616,168.690,37.303,157.010
C06919=1038.435,-69.161,421.604,168.693,37.303,157.010
C06920=1038.441,-68.911,421.593,168.695,37.302,157.010
C06921=1038.448,-68.662,421.581,168.698,37.302,157.010
C06922=1038.454,-68.413,421.570,168.700,37.302,157.010
C06923=1038.460,-68.129,421.556,168.703,37.302,157.010
C06924=1038.467,-67.847,421.543,168.706,37.302,157.010
C06925=1038.474,-67.564,421.530,168.708,37.302,157.010
C06926=1038.481,-67.280,421.516,168.711,37.302,157.010
C06927=1038.487,-67.032,421.505,168.715,37.303,157.010
C06928=1038.494,-66.781,421.494,168.717,37.303,157.010
C06929=1038.500,-66.532,421.482,168.720,37.303,157.010
C06930=1038.506,-66.283,421.469,168.722,37.303,157.010
C06931=1038.512,-66.032,421.458,168.724,37.303,157.010
C06932=1038.519,-65.783,421.446,168.727,37.302,157.010
C06933=1038.525,-65.534,421.435,168.729,37.302,157.010
C06934=1038.530,-65.284,421.423,168.732,37.302,157.010
C06935=1038.537,-65.034,421.411,168.734,37.302,157.010
C06936=1038.543,-64.785,421.399,168.737,37.302,157.010
C06937=1038.549,-64.535,421.387,168.739,37.302,157.010
C06938=1038.555,-64.285,421.375,168.741,37.302,157.010
C06939=1038.562,-64.035,421.363,168.744,37.302,157.010
C06940=1038.568,-63.787,421.352,168.746,37.302,157.010
C06941=1038.573,-63.536,421.340,168.749,37.302,157.010
C06942=1038.580,-63.286,421.328,168.751,37.302,157.010
C06943=1038.587,-63.037,421.316,168.753,37.302,157.010
C06944=1038.592,-62.788,421.304,168.756,37.303,157.010
C06945=1038.598,-62.538,421.293,168.758,37.302,157.010
C06946=1038.605,-62.288,421.281,168.761,37.302,157.010
C06947=1038.612,-62.038,421.269,168.763,37.302,157.010
C06948=1038.617,-61.789,421.257,168.766,37.302,157.010
C06949=1038.624,-61.540,421.245,168.768,37.302,157.010
C06950=1038.630,-61.289,421.233,168.770,37.302,157.010
C06951=1038.636,-61.040,421.221,168.773,37.302,157.010
C06952=1038.642,-60.790,421.209,168.775,37.302,157.010
C06953=1038.649,-60.541,421.197,168.778,37.302,157.010
C06954=1038.654,-60.291,421.185,168.780,37.302,157.010
C06955=1038.661,-60.042,421.173,168.782,37.302,157.010
C06956=1038.667,-59.791,421.162,168.785,37.303,157.011
C06957=1038.674,-59.542,421.150,168.787,37.303,157.011
C06958=1038.680,-59.292,421.137,168.790,37.302,157.011
C06959=1038.686,-59.043,421.125,168.792,37.302,157.011
C06960=1038.693,-58.794,421.113,168.794,37.302,157.011
C06961=1038.699,-58.544,421.101,168.797,37.302,157.011
C06962=1038.705,-58.294,421.089,168.799,37.302,157.011
C06963=1038.712,-58.045,421.077,168.802,37.302,157.011
C06964=1038.718,-57.795,421.064,168.804,37.302,157.011
C06965=1038.724,-57.545,421.052,168.806,37.302,157.011
C06966=1038.730,-57.296,421.041,168.809,37.303,157.011
C06967=1038.736,-57.046,421.028,168.811,37.303,157.011
C06968=1038.743,-56.796,421.017,168.814,37.303,157.011
C06969=1038.749,-56.547,421.005,168.816,37.303,157.011
C06970=1038.755,-56.297,420.993,168.818,37.303,157.011
C06971=1038.762,-56.047,420.981,168.821,37.302,157.011
C06972=1038.769,-55.798,420.969,168.823,37.302,157.011
C06973=1038.774,-55.548,420.956,168.826,37.302,157.011
C06974=1038.781,-55.298,420.944,168.828,37.302,157.011
C06975=1038.787,-55.048,420.932,168.830,37.303,157.011
C06976=1038.794,-54.799,420.920,168.833,37.303,157.011
C06977=1038.800,-54.550,420.907,168.835,37.303,157.011
C06978=1038.806,-54.301,420.895,168.838,37.303,157.011
C06979=1038.813,-54.051,420.883,168.840,37.303,157.011
C06980=1038.819,-53.801,420.871,168.842,37.303,157.011
C06981=1038.825,-53.551,420.858,168.845,37.303,157.011
C06982=1038.832,-53.302,420.846,168.847,37.303,157.011
C06983=1038.838,-53.052,420.834,168.850,37.303,157.011
C06984=1038.844,-52.802,420.822,168.852,37.303,157.011
C06985=1038.851,-52.553,420.810,168.854,37.303,157.011
C06986=1038.857,-52.303,420.797,168.857,37.303,157.011
C06987=1038.865,-52.022,420.783,168.859,37.303,157.011
C06988=1038.872,-51.740,420.770,168.862,37.303,157.011
C06989=1038.879,-51.458,420.755,168.865,37.304,157.011
C06990=1038.886,-51.177,420.742,168.867,37.303,157.011
C06991=1038.892,-50.928,420.730,168.870,37.303,157.011
C06992=1038.899,-50.678,420.718,168.872,37.303,157.011
C06993=1038.905,-50.429,420.705,168.874,37.303,157.011
C06994=1038.911,-50.179,420.692,168.878,37.304,157.012
C06995=1038.918,-49.929,420.680,168.880,37.304,157.012
C06996=1038.924,-49.679,420.668,168.882,37.304,157.012
C06997=1038.930,-49.430,420.654,168.885,37.304,157.012
C06998=1038.936,-49.180,420.642,168.887,37.304,157.012
C06999=1038.943,-48.931,420.630,168.889,37.304,157.012
C07000=1038.949,-48.681,420.617,168.892,37.305,157.012
C07001=1038.955,-48.431,420.604,168.894,37.305,157.012
C07002=1038.961,-48.182,420.592,168.896,37.305,157.012
C07003=1038.968,-47.933,420.579,168.899,37.305,157.012
C07004=1038.973,-47.683,420.566,168.901,37.305,157.012
C07005=1038.979,-47.433,420.554,168.903,37.306,157.012
C07006=1038.986,-47.184,420.541,168.906,37.306,157.012
C07007=1038.992,-46.934,420.529,168.908,37.307,157.012
C07008=1038.998,-46.684,420.516,168.910,37.306,157.012
C07009=1039.004,-46.435,420.503,168.912,37.306,157.012
C07010=1039.011,-46.185,420.491,168.915,37.307,157.012
C07011=1039.018,-45.935,420.478,168.917,37.307,157.012
C07012=1039.024,-45.685,420.465,168.919,37.308,157.013
C07013=1039.030,-45.436,420.452,168.922,37.308,157.013
C07014=1039.037,-45.187,420.439,168.924,37.307,157.013
C07015=1039.042,-44.937,420.427,168.926,37.308,157.013
C07016=1039.048,-44.687,420.414,168.929,37.308,157.013
C07017=1039.055,-44.438,420.401,168.931,37.309,157.013
C07018=1039.061,-44.188,420.389,168.933,37.309,157.013
C07019=1039.067,-43.939,420.376,168.936,37.309,157.013
C07020=1039.073,-43.689,420.363,168.939,37.309,157.013
C07021=1039.080,-43.440,420.350,168.941,37.309,157.013
C07022=1039.086,-43.190,420.337,168.943,37.310,157.013
C07023=1039.093,-42.940,420.324,168.946,37.310,157.013
C07024=1039.099,-42.690,420.312,168.948,37.310,157.013
C07025=1039.105,-42.441,420.299,168.950,37.310,157.013
C07026=1039.111,-42.191,420.286,168.952,37.310,157.013
C07027=1039.118,-41.942,420.273,168.955,37.311,157.013
C07028=1039.124,-41.692,420.261,168.957,37.311,157.013
C07029=1039.130,-41.443,420.247,168.959,37.311,157.014
C07030=1039.137,-41.192,420.235,168.962,37.311,157.014
C07031=1039.143,-40.943,420.221,168.964,37.311,157.014
C07032=1039.150,-40.694,420.209,168.966,37.312,157.014
C07033=1039.156,-40.444,420.196,168.968,37.312,157.014
C07034=1039.162,-40.195,420.183,168.971,37.312,157.014
C07035=1039.168,-39.945,420.170,168.973,37.312,157.014
C07036=1039.175,-39.695,420.157,168.975,37.312,157.014
C07037=1039.181,-39.446,420.145,168.978,37.313,157.014
C07038=1039.188,-39.196,420.131,168.980,37.313,157.014
C07039=1039.194,-38.947,420.118,168.982,37.313,157.014
C07040=1039.200,-38.697,420.106,168.984,37.313,157.014
C07041=1039.206,-38.447,420.092,168.987,37.314,157.014
C07042=1039.213,-38.198,420.079,168.989,37.314,157.014
C07043=1039.219,-37.948,420.066,168.992,37.315,157.014
C07044=1039.225,-37.699,420.053,168.994,37.314,157.014
C07045=1039.231,-37.450,420.040,168.997,37.315,157.015
C07046=1039.237,-37.200,420.027,168.999,37.316,157.015
C07047=1039.244,-36.950,420.013,169.001,37.316,157.015
C07048=1039.250,-36.700,420.000,169.003,37.316,157.015
C07049=1039.256,-36.451,419.987,169.006,37.316,157.015
C07050=1039.262,-36.201,419.974,169.008,37.317,157.015
C07051=1039.269,-35.920,419.959,169.010,37.317,157.015
C07052=1039.276,-35.639,419.944,169.013,37.317,157.015
C07053=1039.283,-35.359,419.929,169.015,37.318,157.015
C07054=1039.290,-35.077,419.914,169.018,37.318,157.015
C07055=1039.296,-34.828,419.901,169.020,37.318,157.015
C07056=1039.303,-34.578,419.887,169.022,37.319,157.016
C07057=1039.309,-34.328,419.874,169.024,37.319,157.016
C07058=1039.315,-34.079,419.862,169.027,37.320,157.016
C07059=1039.321,-33.829,419.848,169.029,37.320,157.016
C07060=1039.328,-33.579,419.835,169.032,37.320,157.016
C07061=1039.334,-33.330,419.821,169.034,37.321,157.016
C07062=1039.341,-33.081,419.808,169.037,37.321,157.016
C07063=1039.347,-32.831,419.794,169.039,37.321,157.016
C07064=1039.354,-32.582,419.781,169.041,37.321,157.016
C07065=1039.360,-32.332,419.769,169.043,37.322,157.016
C07066=1039.366,-32.082,419.755,169.045,37.322,157.016
C07067=1039.372,-31.832,419.741,169.048,37.322,157.016
C07068=1039.378,-31.583,419.728,169.050,37.323,157.017
C07069=1039.384,-31.334,419.715,169.052,37.323,157.017
C07070=1039.391,-31.084,419.701,169.054,37.324,157.017
C07071=1039.397,-30.834,419.688,169.056,37.324,157.017
C07072=1039.404,-30.585,419.674,169.059,37.324,157.017
C07073=1039.410,-30.335,419.661,169.061,37.325,157.017
C07074=1039.417,-30.086,419.648,169.063,37.325,157.017
C07075=1039.423,-29.837,419.634,169.065,37.325,157.017
C07076=1039.430,-29.587,419.621,169.067,37.326,157.017
C07077=1039.436,-29.337,419.607,169.070,37.326,157.017
C07078=1039.442,-29.088,419.594,169.073,37.326,157.017
C07079=1039.448,-28.838,419.580,169.075,37.326,157.017
C07080=1039.454,-28.589,419.567,169.077,37.327,157.017
C07081=1039.461,-28.339,419.553,169.079,37.328,157.018
C07082=1039.467,-28.089,419.540,169.082,37.328,157.018
C07083=1039.474,-27.840,419.526,169.084,37.328,157.018
C07084=1039.480,-27.590,419.513,169.086,37.328,157.018
C07085=1039.487,-27.341,419.500,169.088,37.329,157.018
C07086=1039.493,-27.092,419.486,169.090,37.329,157.018
C07087=1039.499,-26.841,419.472,169.093,37.329,157.018
C07088=1039.505,-26.592,419.459,169.095,37.330,157.018
C07089=1039.512,-26.342,419.445,169.097,37.330,157.018
C07090=1039.517,-26.093,419.431,169.099,37.331,157.018
C07091=1039.524,-25.843,419.418,169.101,37.331,157.018
C07092=1039.530,-25.593,419.404,169.103,37.332,157.019
C07093=1039.536,-25.344,419.390,169.107,37.332,157.019
C07094=1039.543,-25.094,419.376,169.109,37.333,157.019
C07095=1039.549,-24.845,419.363,169.111,37.333,157.019
C07096=1039.555,-24.596,419.349,169.113,37.333,157.019
C07097=1039.562,-24.346,419.335,169.115,37.334,157.019
C07098=1039.568,-24.096,419.322,169.117,37.335,157.019
C07099=1039.574,-23.847,419.307,169.119,37.334,157.019
C07100=1039.580,-23.597,419.294,169.122,37.335,157.019
C07101=1039.587,-23.348,419.281,169.124,37.336,157.019
C07102=1039.593,-23.098,419.266,169.126,37.336,157.020
C07103=1039.599,-22.849,419.252,169.128,37.336,157.020
C07104=1039.605,-22.599,419.238,169.130,37.337,157.020
C07105=1039.611,-22.350,419.225,169.132,37.337,157.020
C07106=1039.618,-22.100,419.211,169.134,37.338,157.020
C07107=1039.624,-21.851,419.197,169.138,37.339,157.020
C07108=1039.631,-21.601,419.183,169.140,37.339,157.020
C07109=1039.637,-21.352,419.170,169.142,37.339,157.020
C07110=1039.643,-21.101,419.156,169.144,37.340,157.020
C07111=1039.650,-20.853,419.142,169.146,37.340,157.021
C07112=1039.656,-20.602,419.127,169.148,37.340,157.021
C07113=1039.662,-20.353,419.114,169.150,37.341,157.021
C07114=1039.669,-20.104,419.100,169.153,37.342,157.021
C07115=1039.676,-19.822,419.085,169.155,37.342,157.021
C07116=1039.683,-19.540,419.069,169.157,37.343,157.021
C07117=1039.690,-19.257,419.053,169.160,37.343,157.021
C07118=1039.697,-18.976,419.037,169.162,37.343,157.021
C07119=1039.703,-18.726,419.023,169.164,37.344,157.021
C07120=1039.710,-18.478,419.009,169.166,37.344,157.021
C07121=1039.716,-18.227,418.995,169.170,37.345,157.022
C07122=1039.723,-17.979,418.981,169.172,37.345,157.022
C07123=1039.729,-17.728,418.967,169.174,37.346,157.022
C07124=1039.735,-17.479,418.953,169.176,37.346,157.022
C07125=1039.742,-17.230,418.939,169.178,37.347,157.022
C07126=1039.748,-16.980,418.925,169.180,37.347,157.022
C07127=1039.755,-16.731,418.911,169.182,37.347,157.022
C07128=1039.761,-16.481,418.897,169.184,37.348,157.022
C07129=1039.767,-16.231,418.883,169.187,37.349,157.022
C07130=1039.774,-15.982,418.869,169.189,37.348,157.022
C07131=1039.779,-15.732,418.855,169.191,37.349,157.023
C07132=1039.787,-15.483,418.841,169.193,37.350,157.023
C07133=1039.793,-15.233,418.827,169.195,37.350,157.023
C07134=1039.799,-14.984,418.813,169.198,37.351,157.023
C07135=1039.805,-14.734,418.798,169.200,37.351,157.023
C07136=1039.811,-14.485,418.784,169.202,37.352,157.023
C07137=1039.818,-14.235,418.770,169.204,37.352,157.023
C07138=1039.824,-13.986,418.756,169.206,37.353,157.023
C07139=1039.830,-13.736,418.741,169.208,37.353,157.023
C07140=1039.837,-13.486,418.727,169.211,37.354,157.024
C07141=1039.843,-13.237,418.712,169.213,37.354,157.024
C07142=1039.849,-12.987,418.698,169.215,37.355,157.024
C07143=1039.855,-12.739,418.684,169.217,37.356,157.024
C07144=1039.862,-12.489,418.669,169.219,37.356,157.024
C07145=1039.868,-12.239,418.655,169.221,37.357,157.024
C07146=1039.874,-11.990,418.641,169.224,37.357,157.024
C07147=1039.880,-11.740,418.627,169.226,37.358,157.024
C07148=1039.886,-11.491,418.612,169.228,37.358,157.024
C07149=1039.893,-11.241,418.598,169.230,37.359,157.025
C07150=1039.899,-10.991,418.584,169.232,37.359,157.025
C07151=1039.905,-10.742,418.569,169.234,37.360,157.025
C07152=1039.912,-10.493,418.555,169.236,37.360,157.025
C07153=1039.918,-10.243,418.541,169.238,37.361,157.025
C07154=1039.924,-9.994,418.526,169.241,37.362,157.025
C07155=1039.931,-9.744,418.512,169.243,37.362,157.025
C07156=1039.937,-9.494,418.497,169.245,37.363,157.026
C07157=1039.943,-9.245,418.483,169.247,37.363,157.026
C07158=1039.950,-8.996,418.468,169.250,37.364,157.026
C07159=1039.957,-8.746,418.453,169.252,37.365,157.026
C07160=1039.962,-8.496,418.440,169.254,37.364,157.026
C07161=1039.969,-8.247,418.425,169.256,37.365,157.026
C07162=1039.976,-7.997,418.410,169.258,37.366,157.026
C07163=1039.981,-7.748,418.396,169.260,37.366,157.026
C07164=1039.988,-7.499,418.382,169.262,37.367,157.026
C07165=1039.995,-7.249,418.367,169.264,37.367,157.027
C07166=1040.000,-7.000,418.353,169.266,37.368,157.027
C07167=1040.007,-6.750,418.338,169.268,37.369,157.027
C07168=1040.013,-6.500,418.324,169.270,37.369,157.027
C07169=1040.020,-6.251,418.309,169.272,37.370,157.027
C07170=1040.026,-6.002,418.294,169.274,37.370,157.027
C07171=1040.033,-5.752,418.280,169.277,37.370,157.027
C07172=1040.039,-5.503,418.265,169.280,37.371,157.027
C07173=1040.046,-5.253,418.250,169.282,37.372,157.027
C07174=1040.052,-5.004,418.237,169.284,37.372,157.028
C07175=1040.058,-4.754,418.222,169.286,37.373,157.028
C07176=1040.065,-4.504,418.207,169.288,37.373,157.028
C07177=1040.071,-4.255,418.192,169.290,37.374,157.028
C07178=1040.077,-4.006,418.178,169.292,37.375,157.028
C07179=1040.085,-3.722,418.161,169.294,37.375,157.028
C07180=1040.092,-3.438,418.145,169.296,37.376,157.028
C07181=1040.099,-3.155,418.127,169.299,37.376,157.028
C07182=1040.106,-2.872,418.111,169.302,37.377,157.029
C07183=1040.112,-2.622,418.096,169.304,37.378,157.029
C07184=1040.119,-2.373,418.081,169.306,37.379,157.029
C07185=1040.124,-2.124,418.067,169.308,37.379,157.029
C07186=1040.131,-1.874,418.052,169.310,37.380,157.029
C07187=1040.137,-1.624,418.037,169.312,37.381,157.029
C07188=1040.144,-1.375,418.022,169.314,37.381,157.030
C07189=1040.149,-1.126,418.007,169.316,37.382,157.030
C07190=1040.156,-0.876,417.992,169.318,37.382,157.030
C07191=1040.162,-0.626,417.977,169.321,37.383,157.030
C07192=1040.169,-0.377,417.962,169.323,37.384,157.030
C07193=1040.174,-0.128,417.948,169.325,37.384,157.030
C07194=1040.180,0.122,417.932,169.327,37.385,157.030
C07195=1040.186,0.372,417.917,169.329,37.386,157.031
C07196=1040.193,0.622,417.902,169.331,37.387,157.031
C07197=1040.199,0.871,417.887,169.333,37.387,157.031
C07198=1040.205,1.120,417.872,169.335,37.388,157.031
C07199=1040.212,1.369,417.857,169.337,37.388,157.031
C07200=1040.218,1.619,417.842,169.339,37.389,157.031
C07201=1040.224,1.869,417.827,169.342,37.390,157.031
C07202=1040.231,2.118,417.812,169.344,37.390,157.031
C07203=1040.237,2.368,417.797,169.346,37.391,157.032
C07204=1040.243,2.617,417.783,169.348,37.391,157.032
C07205=1040.249,2.866,417.768,169.350,37.393,157.032
C07206=1040.256,3.115,417.752,169.352,37.393,157.032
C07207=1040.262,3.365,417.737,169.354,37.394,157.032
C07208=1040.269,3.615,417.722,169.356,37.394,157.032
C07209=1040.275,3.864,417.707,169.357,37.395,157.032
C07210=1040.281,4.113,417.693,169.359,37.396,157.033
C07211=1040.288,4.362,417.677,169.362,37.396,157.033
C07212=1040.293,4.612,417.662,169.364,37.397,157.033
C07213=1040.300,4.862,417.647,169.366,37.397,157.033
C07214=1040.306,5.112,417.632,169.368,37.398,157.033
C07215=1040.312,5.361,417.617,169.370,37.399,157.033
C07216=1040.319,5.610,417.601,169.372,37.399,157.033
C07217=1040.325,5.860,417.586,169.374,37.400,157.034
C07218=1040.332,6.110,417.571,169.376,37.401,157.034
C07219=1040.338,6.359,417.557,169.378,37.402,157.034
C07220=1040.344,6.608,417.541,169.380,37.402,157.034
C07221=1040.351,6.857,417.526,169.383,37.403,157.034
C07222=1040.357,7.107,417.511,169.385,37.403,157.034
C07223=1040.363,7.357,417.496,169.387,37.404,157.034
C07224=1040.369,7.606,417.480,169.389,37.405,157.035
C07225=1040.376,7.856,417.465,169.391,37.405,157.035
C07226=1040.382,8.105,417.450,169.393,37.406,157.035
C07227=1040.389,8.354,417.434,169.395,37.406,157.035
C07228=1040.395,8.604,417.419,169.397,37.407,157.035
C07229=1040.402,8.854,417.404,169.399,37.407,157.035
C07230=1040.408,9.103,417.389,169.401,37.409,157.035
C07231=1040.415,9.352,417.374,169.404,37.409,157.036
C07232=1040.421,9.602,417.359,169.406,37.410,157.036
C07233=1040.428,9.851,417.343,169.408,37.411,157.036
C07234=1040.433,10.101,417.328,169.410,37.411,157.036
C07235=1040.440,10.351,417.313,169.412,37.412,157.036
C07236=1040.446,10.600,417.297,169.414,37.412,157.036
C07237=1040.453,10.849,417.282,169.416,37.413,157.036
C07238=1040.460,11.098,417.266,169.417,37.414,157.036
C07239=1040.466,11.348,417.251,169.419,37.414,157.037
C07240=1040.472,11.598,417.236,169.421,37.415,157.037
C07241=1040.479,11.847,417.221,169.423,37.415,157.037
C07242=1040.485,12.097,417.205,169.426,37.416,157.037
C07243=1040.492,12.382,417.188,169.429,37.416,157.037
C07244=1040.500,12.667,417.170,169.431,37.418,157.037
C07245=1040.507,12.952,417.152,169.433,37.418,157.037
C07246=1040.514,13.238,417.135,169.435,37.419,157.038
C07247=1040.521,13.487,417.120,169.437,37.419,157.038
C07248=1040.528,13.737,417.105,169.439,37.420,157.038
C07249=1040.534,13.986,417.089,169.441,37.421,157.038
C07250=1040.540,14.236,417.073,169.443,37.421,157.038
C07251=1040.547,14.485,417.058,169.446,37.422,157.038
C07252=1040.553,14.735,417.043,169.448,37.423,157.039
C07253=1040.559,14.984,417.027,169.450,37.424,157.039
C07254=1040.566,15.233,417.011,169.452,37.424,157.039
C07255=1040.574,15.563,416.991,169.454,37.425,157.039
C07256=1040.582,15.892,416.969,169.457,37.426,157.039
C07257=1040.590,16.223,416.949,169.459,37.427,157.039
C07258=1040.599,16.552,416.929,169.463,37.428,157.040
C07259=1040.605,16.802,416.913,169.465,37.429,157.040
C07260=1040.611,17.051,416.897,169.467,37.430,157.040
C07261=1040.618,17.301,416.882,169.468,37.430,157.040
C07262=1040.624,17.550,416.866,169.470,37.431,157.040
C07263=1040.630,17.799,416.850,169.472,37.432,157.040
C07264=1040.637,18.049,416.835,169.474,37.433,157.041
C07265=1040.643,18.298,416.819,169.476,37.433,157.041
C07266=1040.649,18.547,416.803,169.478,37.434,157.041
C07267=1040.656,18.797,416.788,169.480,37.434,157.041
C07268=1040.662,19.047,416.772,169.483,37.435,157.041
C07269=1040.669,19.296,416.756,169.485,37.436,157.041
C07270=1040.675,19.546,416.740,169.487,37.437,157.041
C07271=1040.681,19.795,416.725,169.489,37.437,157.042
C07272=1040.688,20.044,416.709,169.490,37.438,157.042
C07273=1040.694,20.293,416.693,169.492,37.439,157.042
C07274=1040.700,20.543,416.677,169.494,37.440,157.042
C07275=1040.706,20.792,416.662,169.496,37.440,157.042
C07276=1040.712,21.041,416.645,169.498,37.441,157.042
C07277=1040.720,21.291,416.629,169.501,37.442,157.042
C07278=1040.725,21.541,416.614,169.503,37.443,157.043
C07279=1040.732,21.790,416.598,169.505,37.443,157.043
C07280=1040.738,22.040,416.582,169.506,37.444,157.043
C07281=1040.745,22.289,416.566,169.508,37.445,157.043
C07282=1040.750,22.538,416.550,169.510,37.446,157.043
C07283=1040.757,22.787,416.534,169.512,37.447,157.043
